RoboDK station: reto.rdk

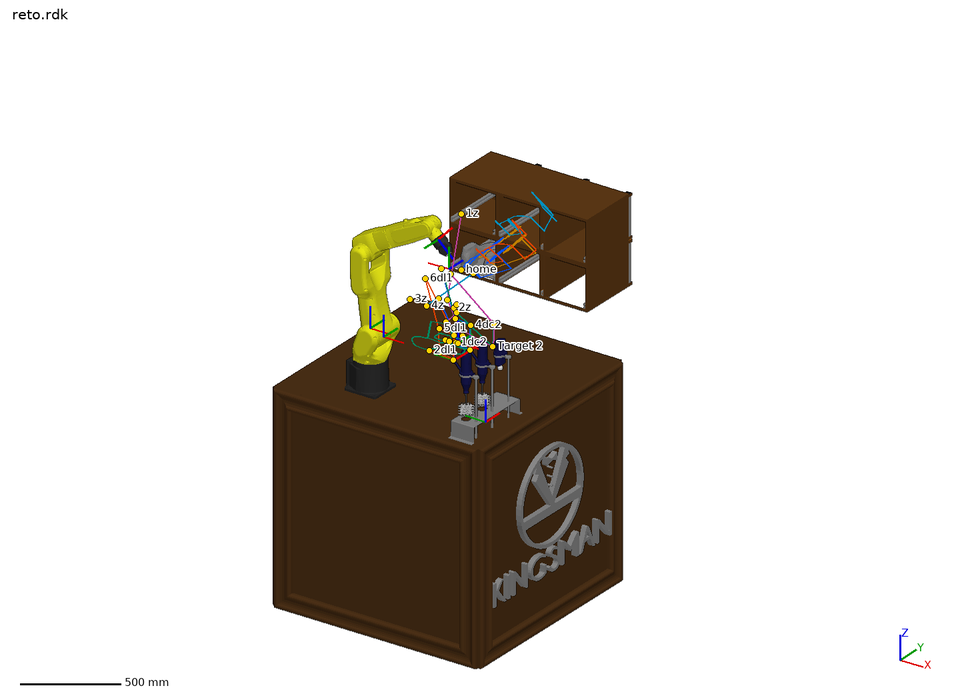
[picture v0: the station drawn from its stored meshes, robots at their saved joint values, targets as dots, program paths as lines]
Station reto (saved by RoboDK 5.5.4). Poses are relative to the parent item; angles as X-Y-Z fixed-axis rotations.
  - frame Fanuc LR Mate 200iD/7L Base at (0, 670, 330) mm
    - robot Fanuc LR Mate 200iD/7L: 6 axes, payload 7 kg, reach 911 mm, repeatability 0.03 mm, weight 27 kg
        modified DH rows (alpha deg, a mm, theta deg, d mm): 0, 0, 0, 330; -90, 50, -90, 0; 0, 440, 0, 0; -90, 35, 0, 420; 90, 0, 0, 0; -90, 0, 0, 80
        base shift (0, 0, -330) mm
        joint limits [-170, -70, -70, -190, -115, -360] to [170, 145, 215, 190, 115, 360]; home [0, 0, 0, 0, 0, 0]; saved at [0, -7.035, 27.253, 0, -70.54, 0]
      - frame RobotiQ 2F-140 Gripper (Mechanism) Base at (0, 0, 0) mm
        - robot RobotiQ 2F-140 Gripper (Mechanism) (model RobotiQ 2F140): 1 axes, payload 5 kg
            joint limits [0] to [140]; home [140]; saved at [30]
          - tool Tool 1, TCP at (0, 0, 190) mm
        - target open (joint target) at (0, 0, 190) mm; joints [30] of RobotiQ 2F-140 Gripper (Mechanism)
        - target close (joint target) at (-70.03, -6.66, -1.07) mm, rotated rx -1.32 ry 1.53 rz 3.85 deg; joints [10] of RobotiQ 2F-140 Gripper (Mechanism)
    - target home (Cartesian target) at (550, 0, 475) mm, rotated rx -180 ry -46.71 rz 0 deg; joints [0, 3.939, 7.691, 0, -50.978, 0] of Fanuc LR Mate 200iD/7L
  - frame rack at (-170, 1590, 240) mm, rotated rx 90 ry 0 rz 180 deg
    - object FullRack (1) at (-810, 360, -320) mm, size 835 x 510 x 385.3 mm, geometry from FullRack (1).STEP
    - target 1z (Cartesian target) at (-358.1, 564.97, -403.2) mm, rotated rx -26.57 ry -40.12 rz 107.86 deg; joints [70, -7.04, 27.25, 0, -70.54, 0] of Fanuc LR Mate 200iD/7L
    - target 2z (Cartesian target) at (-342.39, 58.73, -444.89) mm, rotated rx 2.43 ry -28.49 rz 101.39 deg; joints [48.708, 3.516, -60.085, -111.282, -47, 134.319] of Fanuc LR Mate 200iD/7L
    - target 3z (Cartesian target) at (-104.58, 56.68, -482.72) mm, rotated rx 2.43 ry -28.49 rz 101.39 deg; joints [97.474, -14.415, -55.536, -177.531, -28.246, 164.28] of Fanuc LR Mate 200iD/7L
    - target 4z (Cartesian target) at (-165.76, 16.78, -430.34) mm, rotated rx 2.43 ry -28.49 rz 101.39 deg; joints [82.687, 5.107, -71.647, -159.69, -45.234, 158.787] of Fanuc LR Mate 200iD/7L
    - target 5z (Cartesian target) at (-150, 20, 0) mm, rotated rx 2.43 ry -28.49 rz 101.39 deg; joints [88.603, 43.78, -43.517, 30.239, 18.18, -38.415] of Fanuc LR Mate 200iD/7L
    - target subida charola (Cartesian target) at (-343.88, 69.1, -423.53) mm, rotated rx 2.43 ry -28.49 rz 101.39 deg; joints [50.933, 3.87, -57.639, 68.607, 45.039, -48.263] of Fanuc LR Mate 200iD/7L
  - frame base herramental at (710, 650, 20) mm, rotated rx 0 ry 0 rz 90 deg
    - object Soporte de herramientas at (0, 0, 70) mm, rotated rx 90 ry 0 rz 180 deg, size 443.6 x 340 x 140 mm, geometry from Soporte de herramientas.STEP
  - frame dremel2 at (620, 650, 390) mm, rotated rx 0 ry 0 rz 90 deg
    - target 1dc2 (Cartesian target) at (0.49, 88.9, 17.55) mm, rotated rx -180 ry -61.75 rz -90 deg; joints [89.913, -3.297, -48.984, 180.078, 102.766, 0.058] of Fanuc LR Mate 200iD/7L
    - target 2dc2 (Cartesian target) at (0, 151.76, 13.3) mm, rotated rx -180 ry -61.75 rz -90 deg; joints [-4.961, -25.961, -32.248, 48.26, 5.86, -45.758] of Fanuc LR Mate 200iD/7L
    - target 3dc2 (Cartesian target) at (0, 4.92, 1.2) mm, rotated rx -180 ry -49.6 rz -90 deg; joints [-2.796, -1.172, -33.671, 162.466, 7.084, -160.778] of Fanuc LR Mate 200iD/7L
    - target 4dc2 (Cartesian target) at (0, 0.76, 138.38) mm, rotated rx -180 ry -49.6 rz -90 deg; joints [-2.768, -6.859, -13.429, 175.365, 27.075, -174.076] of Fanuc LR Mate 200iD/7L
    - target 5dc2 (Cartesian target) at (0, 92.68, 148.84) mm, rotated rx -180 ry -44.51 rz -90 deg; joints [-3.386, -17.516, -7.24, 176.175, 38.363, -174.583] of Fanuc LR Mate 200iD/7L
    - target 6dc2 (Cartesian target) at (477.83, 510, 116.81) mm, rotated rx -180 ry -49.6 rz 3.55 deg; joints [64.081, -25.306, -11.026, 143.659, 39.225, -130.203] of Fanuc LR Mate 200iD/7L
  - frame dremel1 at (620, 510.31, 389.97) mm, rotated rx 0 ry 0 rz 90 deg
    - target 1dl1 (Cartesian target) at (0.49, 88.9, 17.55) mm, rotated rx -180 ry -61.75 rz -90 deg; joints [-28.495, -9.165, -37.687, 76.78, 25.575, -60.993] of Fanuc LR Mate 200iD/7L
    - target 2dl1 (Cartesian target) at (0, 151.76, 13.3) mm, rotated rx -180 ry -61.75 rz -90 deg; joints [-34.725, -17.114, -36.143, 84.899, 30.251, -65.939] of Fanuc LR Mate 200iD/7L
    - target 3dl1 (Cartesian target) at (0, 4.92, 1.2) mm, rotated rx -180 ry -49.6 rz -90 deg; joints [-21.306, 2.651, -33.616, 117.955, 18.257, -105.014] of Fanuc LR Mate 200iD/7L
    - target 4dl1 (Cartesian target) at (0, 0.76, 138.38) mm, rotated rx -180 ry -48.03 rz -90 deg; joints [-20.886, -2.493, -13.042, 151.816, 34.141, -141.769] of Fanuc LR Mate 200iD/7L
    - target 5dl1 (Cartesian target) at (0, 92.68, 148.84) mm, rotated rx -180 ry -49.6 rz -90 deg; joints [-26.4, -14.504, -10.508, 146.56, 37.916, -134.648] of Fanuc LR Mate 200iD/7L
    - target 6dl1 (Cartesian target) at (477.83, 510, 116.81) mm, rotated rx -180 ry -55.33 rz 3.55 deg; joints [37.94, -45.517, -1.764, 129.234, 61.201, -109.727] of Fanuc LR Mate 200iD/7L
    - object cepillo1 at (0, -70, -50) mm, rotated rx 90 ry 0 rz 180 deg, size 80 x 351.1 x 124.1 mm, geometry from Dremel con brida.STEP
  - frame bote cera at (140, 586, 355) mm
    - target Target 1 (Cartesian target) at (316.19, 84, 136.54) mm, rotated rx -180 ry -46.71 rz 0 deg; joints [0, -28.492, -10.215, 0, -33.072, 0] of Fanuc LR Mate 200iD/7L
    - target Target 3 (Cartesian target) at (300.65, 202.07, 136.5) mm, rotated rx -180 ry -46.9 rz 15 deg; joints [15, -28.576, -10.266, 0, -32.834, 0] of Fanuc LR Mate 200iD/7L
    - target Target 2 (Cartesian target) at (513.63, 208.92, 6.17) mm, rotated rx -180 ry -50.56 rz 10.82 deg; joints [10.82, 7.34, -38.44, 0, -1, 0] of Fanuc LR Mate 200iD/7L
    - target Target 4 (Cartesian target) at (516.39, 216.06, 127.59) mm, rotated rx -179.95 ry -49.71 rz 10.96 deg; joints [11.533, 0.978, -20.278, 1.139, -20.021, -1.442] of Fanuc LR Mate 200iD/7L
    - target Target 5 (Cartesian target) at (-30, 622.41, 89.17) mm, rotated rx -179.99 ry -46.7 rz 79.99 deg; joints [77.59, -12.853, -22.678, -4.973, -20.717, 6.303] of Fanuc LR Mate 200iD/7L
  - program open (3 instructions, listed below)
  - program close (3 instructions, listed below)
  - program home (4 instructions, listed below)
  - object mesa at (-1220, 1130, 330) mm, size 1277.5 x 1274.9 x 1205 mm, geometry from mesa.STEP
  - frame zapato at (110, 1270, 40) mm
    - target Target 1 (Cartesian target) at (78.1, -83.2, 764.97) mm, rotated rx -180 ry -46.71 rz 70 deg; joints [70, -7.04, 27.25, 0, -70.54, 0] of Fanuc LR Mate 200iD/7L
    - target Target 2 (Cartesian target) at (48.8, -163.69, 316.74) mm, rotated rx 180 ry -45.09 rz 70 deg; joints [70, -19.91, -32.531, 0, -12.378, 0] of Fanuc LR Mate 200iD/7L
    - target Target 3 (Cartesian target) at (51.99, -36.78, 68.56) mm, rotated rx -154.66 ry -59.5 rz 70 deg; joints [58.654, 42.845, -90.321, 40.028, 62.94, -13.915] of Fanuc LR Mate 200iD/7L
    - target Target 4 (Cartesian target) at (0, 0, 0) mm, rotated rx -154.66 ry -59.5 rz 70 deg; joints [67.996, 54.587, -97.1, 29.193, 68.847, -10.257] of Fanuc LR Mate 200iD/7L
    - target Target 5 (Cartesian target) at (-12.96, -146.91, 298.71) mm, rotated rx -168.48 ry -59.46 rz 67.92 deg; joints [74.53, -18.6, -45.29, -158.86, -16.3, 156.27] of Fanuc LR Mate 200iD/7L
    - target Target 6 (Cartesian target) at (14.48, -93.65, 48.92) mm, rotated rx -154.66 ry -59.5 rz 70 deg; joints [59.102, 46.97, -102.654, -143.53, -72.674, 174.279] of Fanuc LR Mate 200iD/7L
  - program recoger cepillo cera (10 instructions, listed below)
  - program reset (1 instructions, listed below)
  - program recoger cepillo limpieza (10 instructions, listed below)
  - program recoger cera (9 instructions, listed below)
  - program pick charola (8 instructions, listed below)
  - program c1 recoger (7 instructions, listed below)
  - program c1 entregar (7 instructions, listed below)
  - program poscharolamesa (7 instructions, listed below)
  - program dejar cepillo limpieza (9 instructions, listed below)
  - program dejar cepillo cera (10 instructions, listed below)
  - program dejar  cera (9 instructions, listed below)
  - program rutinac1 (22 instructions, listed below)
  - machining project parribaizq: rotZ(0) | rotX(0)*rotY(0) | onStart | onPathStart | onApproach | onPoint | onRetract | onFinish | SetRPM(%1) | SetTool(%1) | Extruder(%1) | default | default | OutOnMov(%1) | OutOffMov(%1) | onPathFinish | M_RunCode(%1)
  - program platizq (163 instructions, listed below)
  - machining project plateralesizq: rotZ(0) | rotX(0)*rotY(0) | onStart | onPathStart | onApproach | onPoint | onRetract | onFinish | SetRPM(%1) | SetTool(%1) | Extruder(%1) | default | default | OutOnMov(%1) | OutOffMov(%1) | onPathFinish | M_RunCode(%1)
  - program parrizq (66 instructions, listed below)
  - machining project Path3 ajustes: rotZ(0) | rotX(0)*rotY(0) | onStart | onPathStart | onApproach | onPoint | onRetract | onFinish | SetRPM(%1) | SetTool(%1) | Extruder(%1) | default | default | OutOnMov(%1) | OutOffMov(%1) | onPathFinish | M_RunCode(%1)
  - program platder (154 instructions, listed below)
  - machining project Path4 ajustes: rotZ(0) | rotX(0)*rotY(0) | onStart | onPathStart | onApproach | onPoint | onRetract | onFinish | SetRPM(%1) | SetTool(%1) | Extruder(%1) | default | default | OutOnMov(%1) | OutOffMov(%1) | onPathFinish | M_RunCode(%1)
  - program parrder (59 instructions, listed below)
  - object zapatoconcharola at (-21.13, 1591.46, 262.04) mm, rotated rx 0 ry 0 rz -0.01 deg, size 250 x 350 x 100.5 mm, geometry from zapatoconcharola.STEP
    - object Ruta_IZQ at (-60, 470, 60) mm, rotated rx 0 ry 0 rz -90 deg, geometry from Curva importada
    - object R7 at (-105, 460, 60) mm, rotated rx 0 ry 0 rz -90 deg
  - object cepillo2 at (690, 650, 340) mm, rotated rx 90 ry 0 rz -90 deg, size 80 x 351.1 x 124.1 mm, geometry from Dremel con brida.STEP
  - machining project Path5 ajustes: rotZ(0) | rotX(0)*rotY(0) | onStart | onPathStart | onApproach | onPoint | onRetract | onFinish | SetRPM(%1) | SetTool(%1) | Extruder(%1) | default | default | OutOnMov(%1) | OutOffMov(%1) | onPathFinish | M_RunCode(%1)
  - program Path5 (163 instructions, listed below)
  - object Bote con brida at (698, 771, 410) mm, rotated rx 90 ry 0 rz -90 deg, size 75 x 160 x 85 mm, geometry from Bote con brida.STEP
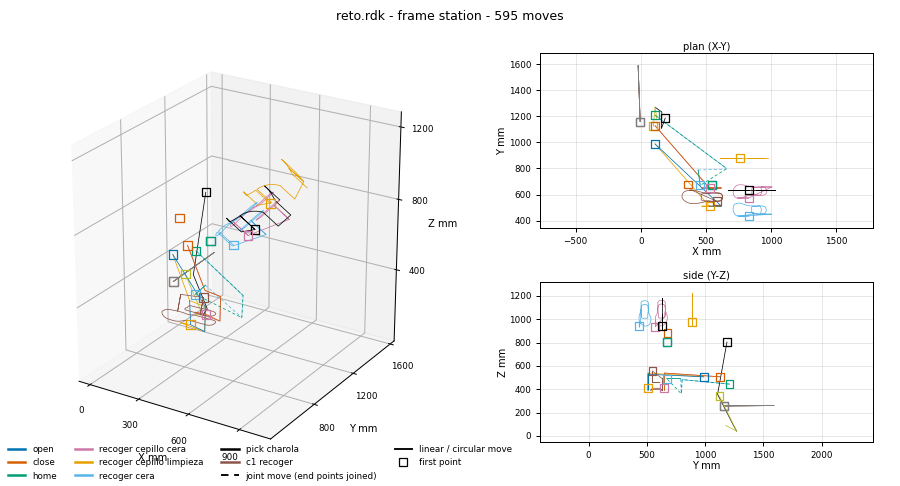
[picture p0: tool path of reto.rdk in frame station, 595 of 595 moves have a stored position in this frame; points joined in program order, loops and branches not executed]

--- program open (robot RobotiQ 2F-140 Gripper (Mechanism)) ---
  Est. Ref.: RobotiQ 2F-140 Gripper (Mechanism) Base
  Est. herr: Tool 1
  MoveJ (open)

--- program close (robot RobotiQ 2F-140 Gripper (Mechanism)) ---
  Est. Ref.: RobotiQ 2F-140 Gripper (Mechanism) Base
  Est. herr: Tool 1
  MoveJ (close)

--- program home (robot Fanuc LR Mate 200iD/7L) ---
  Est. Ref.: Fanuc LR Mate 200iD/7L Base
  MoveJ (home)
  Llamar open
  Separar de Tool 1

--- program recoger cepillo cera (robot Fanuc LR Mate 200iD/7L) ---
  Est. Ref.: dremel2
  Est. herr: Tool 1
  MoveL (1dc2)
  MoveL (Target 2) -> target 2dc2
  MoveL (Target 3) -> target 3dc2
  Llamar close
  Adjuntar a Tool 1
  MoveL (Target 4) -> target 4dc2
  MoveL (Target 5) -> target 5dc2
  MoveL (6dc2)

--- program reset (robot Fanuc LR Mate 200iD/7L) ---
  Reemplazar objetos

--- program recoger cepillo limpieza (robot Fanuc LR Mate 200iD/7L) ---
  Est. Ref.: dremel1
  Est. herr: Tool 1
  MoveL (1dl1)
  MoveL (2dl1)
  MoveL (3dl1)
  Adjuntar a Tool 1
  Llamar close
  MoveL (4dl1)
  MoveL (5dl1)
  MoveL (6dl1)

--- program recoger cera (robot Fanuc LR Mate 200iD/7L) ---
  Est. Ref.: bote cera
  Est. herr: Tool 1
  MoveJ (Target 1)
  MoveL (Target 3)
  MoveJ (Target 2)
  Llamar close
  Adjuntar a Tool 1
  MoveJ (Target 4)
  MoveL (Target 5)

--- program pick charola (robot Fanuc LR Mate 200iD/7L) ---
  Est. Ref.: zapato
  Est. herr: Tool 1
  MoveJ (Target 1)
  MoveL (Target 2)
  MoveL (Target 3)
  MoveL (Target 4)
  Llamar close
  Adjuntar a Tool 1

--- program c1 recoger (robot Fanuc LR Mate 200iD/7L) ---
  Est. Ref.: rack
  Est. herr: Tool 1
  MoveL (4z)
  MoveL (Target 4) -> target 5z
  Adjuntar a Tool 1
  Llamar close
  MoveL (4z)

--- program c1 entregar (robot Fanuc LR Mate 200iD/7L) ---
  Est. Ref.: rack
  Est. herr: Tool 1
  MoveL (4z)
  MoveL (Target 4) -> target 5z
  Separar de Tool 1
  Llamar open
  MoveL (4z)

--- program poscharolamesa (robot Fanuc LR Mate 200iD/7L) ---
  Est. Ref.: zapato
  Est. herr: Tool 1
  MoveJ (Target 5)
  MoveL (Target 4)
  Separar de Tool 1
  Llamar open
  MoveL (Target 6)

--- program dejar cepillo limpieza (robot Fanuc LR Mate 200iD/7L) ---
  Est. Ref.: dremel1
  Est. herr: Tool 1
  MoveL (6dl1)
  MoveL (4dl1)
  MoveL (3dl1)
  Separar de Tool 1
  Llamar open
  MoveL (1dl1)
  MoveL (5dl1)

--- program dejar cepillo cera (robot Fanuc LR Mate 200iD/7L) ---
  Est. Ref.: dremel2
  Est. herr: Tool 1
  MoveL (6dc2)
  MoveL (Target 5) -> target 5dc2
  MoveL (Target 4) -> target 4dc2
  MoveL (Target 3) -> target 3dc2
  Llamar open
  Separar de Tool 1
  MoveL (1dc2)
  MoveL (Target 2) -> target 2dc2

--- program dejar  cera (robot Fanuc LR Mate 200iD/7L) ---
  Est. Ref.: bote cera
  Est. herr: Tool 1
  MoveL (Target 5)
  MoveJ (Target 4)
  MoveJ (Target 2)
  Llamar open
  Separar de Tool 1
  MoveJ (Target 1)
  MoveL (Target 3)

--- program rutinac1 (robot Fanuc LR Mate 200iD/7L) ---
  Llamar home
  Llamar c1 recoger
  Llamar poscharolamesa
  Llamar home
  Llamar recoger cera
  Llamar recoger cepillo cera
  Llamar platizq
  Llamar parrizq
  Llamar platder
  Llamar parrder
  Llamar dejar cepillo cera
  Llamar recoger cepillo limpi...: recoger cepillo limpieza
  Llamar platizq
  Llamar parrizq
  Llamar platder
  Llamar parrder
  Llamar dejar cepillo limpieza
  Llamar Program1
  Llamar pick charola
  Llamar pos entrega
  Llamar c1 entregar
  Llamar home

--- program platizq (robot Fanuc LR Mate 200iD/7L) ---
  Suave(1)
  Establecer velocidad (1000.0 mm/s)
  Est. Ref.: RobotiQ 2F-140 Gripper (Mechanism) Base
  Est. herr: Tool 1
  Mostrar Tool 1
  MoveJ 1 to (286.31, 96.93, 301.9) mm, rotated rx 164.21 ry -43.9 rz -78.89 deg; joints [65.752, 52.412, -5.749, -44.813, -95.376, 119.1]
  MoveL 2 to (286.31, 96.93, 301.9) mm, rotated rx 164.21 ry -43.9 rz -78.89 deg; joints [65.752, 52.412, -5.749, -44.813, -95.376, 119.1]
  MoveL 3 to (266.7, 96.93, 203.84) mm, rotated rx 164.21 ry -43.9 rz -78.89 deg; joints [66.303, 57.855, -14.466, -44.7, -88.799, 124.852]
  MoveL 4 to (266.7, 96.93, 203.84) mm, rotated rx 164.21 ry -43.9 rz -78.89 deg; joints [66.303, 57.855, -14.466, -44.7, -88.799, 124.852]
  Establecer velocidad (50.0 mm/s)
  MoveL 5 to (278.42, 97.92, 203.84) mm, rotated rx 164.21 ry -43.9 rz -78.89 deg; joints [65.914, 55.94, -16.17, -44.64, -87.851, 126.317]
  MoveL 6 to (290.23, 97.9, 203.84) mm, rotated rx 164.21 ry -43.9 rz -78.89 deg; joints [65.577, 54.073, -17.804, -44.604, -86.914, 127.696]
  MoveL 7 to (301.99, 96.89, 203.84) mm, rotated rx 164.21 ry -43.9 rz -78.89 deg; joints [65.297, 52.255, -19.368, -44.595, -85.987, 128.985]
  MoveL 8 to (313.58, 94.89, 203.84) mm, rotated rx 164.21 ry -43.9 rz -78.89 deg; joints [65.079, 50.491, -20.859, -44.613, -85.069, 130.182]
  MoveL 9 to (324.92, 91.93, 204.39) mm, rotated rx 164.21 ry -43.9 rz -78.89 deg; joints [64.926, 48.755, -22.224, -44.657, -84.197, 131.247]
  MoveL 10 to (336.63, 87.99, 206.05) mm, rotated rx 164.21 ry -43.9 rz -78.89 deg; joints [64.822, 46.928, -23.474, -44.719, -83.376, 132.199]
  MoveL 11 to (348.23, 84.53, 208.85) mm, rotated rx 164.21 ry -43.9 rz -78.89 deg; joints [64.687, 45.145, -24.49, -44.762, -82.742, 133.009]
  MoveL 12 to (359.72, 81.7, 212.77) mm, rotated rx 164.21 ry -43.9 rz -78.89 deg; joints [64.506, 43.399, -25.277, -44.774, -82.298, 133.685]
  MoveL 13 to (371.38, 79.44, 216.26) mm, rotated rx 164.21 ry -43.9 rz -78.89 deg; joints [64.274, 41.719, -26.039, -44.769, -81.905, 134.376]
  MoveL 14 to (383.33, 77.72, 218.59) mm, rotated rx 164.21 ry -43.9 rz -78.89 deg; joints [63.986, 40.127, -26.87, -44.752, -81.496, 135.153]
  MoveL 15 to (395.57, 76.59, 219.75) mm, rotated rx 164.21 ry -43.9 rz -78.89 deg; joints [63.637, 38.623, -27.777, -44.724, -81.07, 136.022]
  MoveL 16 to (408.89, 76.07, 219.88) mm, rotated rx 164.21 ry -43.9 rz -78.89 deg; joints [63.191, 37.12, -28.809, -44.675, -80.612, 137.04]
  MoveL 17 to (422.22, 76.27, 219.88) mm, rotated rx 164.21 ry -43.9 rz -78.89 deg; joints [62.676, 35.694, -29.78, -44.591, -80.237, 138.056]
  MoveL 18 to (435.55, 76.27, 219.88) mm, rotated rx 164.21 ry -43.9 rz -78.89 deg; joints [62.158, 34.286, -30.714, -44.501, -79.885, 139.045]
  MoveL 19 to (448.88, 76.27, 219.88) mm, rotated rx 164.21 ry -43.9 rz -78.89 deg; joints [61.622, 32.904, -31.606, -44.396, -79.57, 140.012]
  MoveL 20 to (462.2, 76.27, 219.88) mm, rotated rx 164.21 ry -43.9 rz -78.89 deg; joints [61.067, 31.545, -32.457, -44.276, -79.291, 140.96]
  MoveL 21 to (470.53, 76.27, 219.88) mm, rotated rx 164.21 ry -43.9 rz -78.89 deg; joints [60.709, 30.706, -32.969, -44.192, -79.133, 141.543]
  MoveL 22 to (478.87, 76.27, 219.88) mm, rotated rx 164.21 ry -43.9 rz -78.89 deg; joints [60.344, 29.875, -33.467, -44.101, -78.989, 142.119]
  MoveL 23 to (487.2, 76.27, 219.88) mm, rotated rx 164.21 ry -43.9 rz -78.89 deg; joints [59.97, 29.052, -33.95, -44.003, -78.858, 142.689]
  MoveL 24 to (495.6, 76.03, 219.88) mm, rotated rx 164.21 ry -43.9 rz -78.89 deg; joints [59.603, 28.214, -34.431, -43.906, -78.722, 143.252]
  MoveL 25 to (501.43, 74.59, 219.88) mm, rotated rx 164.21 ry -43.9 rz -78.89 deg; joints [59.445, 27.564, -34.797, -43.886, -78.549, 143.607]
  MoveL 26 to (507.05, 71.76, 219.88) mm, rotated rx 164.21 ry -43.9 rz -78.89 deg; joints [59.406, 26.856, -35.188, -43.924, -78.289, 143.907]
  MoveL 27 to (511.98, 67.62, 219.88) mm, rotated rx 164.21 ry -43.9 rz -78.89 deg; joints [59.506, 26.142, -35.574, -44.026, -77.955, 144.121]
  MoveL 28 to (515.8, 62.47, 219.88) mm, rotated rx 164.21 ry -43.9 rz -78.89 deg; joints [59.745, 25.481, -35.925, -44.188, -77.568, 144.228]
  MoveL 29 to (518.26, 56.77, 219.88) mm, rotated rx 164.21 ry -43.9 rz -78.89 deg; joints [60.1, 24.923, -36.215, -44.397, -77.16, 144.226]
  MoveL 30 to (519.36, 50.99, 219.88) mm, rotated rx 164.21 ry -43.9 rz -78.89 deg; joints [60.532, 24.497, -36.433, -44.631, -76.76, 144.128]
  MoveL 31 to (519.45, 45.42, 219.88) mm, rotated rx 164.21 ry -43.9 rz -78.89 deg; joints [61, 24.185, -36.591, -44.872, -76.383, 143.967]
  MoveL 32 to (519.45, 39.87, 219.88) mm, rotated rx 164.21 ry -43.9 rz -78.89 deg; joints [61.476, 23.887, -36.74, -45.116, -76.008, 143.798]
  MoveL 33 to (518.9, 34.19, 219.88) mm, rotated rx 164.21 ry -43.9 rz -78.89 deg; joints [61.991, 23.64, -36.863, -45.373, -75.629, 143.588]
  MoveL 34 to (517.05, 28.4, 219.88) mm, rotated rx 164.21 ry -43.9 rz -78.89 deg; joints [62.579, 23.523, -36.921, -45.651, -75.253, 143.29]
  MoveL 35 to (513.81, 22.95, 219.88) mm, rotated rx 164.21 ry -43.9 rz -78.89 deg; joints [63.202, 23.567, -36.898, -45.928, -74.911, 142.915]
  MoveL 36 to (509.33, 18.32, 219.88) mm, rotated rx 164.21 ry -43.9 rz -78.89 deg; joints [63.805, 23.785, -36.791, -46.178, -74.638, 142.487]
  MoveL 37 to (503.95, 14.89, 219.88) mm, rotated rx 164.21 ry -43.9 rz -78.89 deg; joints [64.336, 24.157, -36.605, -46.377, -74.459, 142.042]
  MoveL 38 to (498.15, 12.84, 219.88) mm, rotated rx 164.21 ry -43.9 rz -78.89 deg; joints [64.757, 24.644, -36.358, -46.512, -74.384, 141.614]
  MoveL 39 to (490.56, 12.13, 219.88) mm, rotated rx 164.21 ry -43.9 rz -78.89 deg; joints [65.128, 25.38, -35.977, -46.596, -74.428, 141.114]
  MoveL 40 to (483.15, 12.13, 219.88) mm, rotated rx 164.21 ry -43.9 rz -78.89 deg; joints [65.422, 26.134, -35.578, -46.642, -74.529, 140.643]
  MoveL 41 to (475.75, 12.13, 219.88) mm, rotated rx 164.21 ry -43.9 rz -78.89 deg; joints [65.71, 26.891, -35.168, -46.682, -74.64, 140.166]
  MoveL 42 to (468.34, 12.13, 219.88) mm, rotated rx 164.21 ry -43.9 rz -78.89 deg; joints [65.992, 27.653, -34.747, -46.717, -74.761, 139.684]
  MoveL 43 to (460.94, 12.13, 219.88) mm, rotated rx 164.21 ry -43.9 rz -78.89 deg; joints [66.268, 28.419, -34.314, -46.745, -74.892, 139.196]
  MoveL 44 to (453.53, 12.13, 219.88) mm, rotated rx 164.21 ry -43.9 rz -78.89 deg; joints [66.537, 29.189, -33.869, -46.768, -75.034, 138.702]
  MoveL 45 to (438.87, 12.13, 219.88) mm, rotated rx 164.21 ry -43.9 rz -78.89 deg; joints [67.055, 30.73, -32.954, -46.798, -75.346, 137.706]
  MoveL 46 to (424.21, 12.13, 219.88) mm, rotated rx 164.21 ry -43.9 rz -78.89 deg; joints [67.551, 32.293, -31.991, -46.81, -75.7, 136.685]
  MoveL 47 to (409.55, 11.64, 219.88) mm, rotated rx 164.21 ry -43.9 rz -78.89 deg; joints [68.066, 33.859, -30.992, -46.82, -76.064, 135.624]
  MoveL 48 to (394.97, 10.16, 219.72) mm, rotated rx 164.21 ry -43.9 rz -78.89 deg; joints [68.635, 35.412, -29.992, -46.848, -76.39, 134.528]
  MoveL 49 to (382.83, 8.14, 218.52) mm, rotated rx 164.21 ry -43.9 rz -78.89 deg; joints [69.153, 36.756, -29.261, -46.901, -76.56, 133.663]
  MoveL 50 to (370.99, 5.48, 216.16) mm, rotated rx 164.21 ry -43.9 rz -78.89 deg; joints [69.696, 38.124, -28.661, -46.982, -76.623, 132.878]
  MoveL 51 to (359.45, 2.34, 212.67) mm, rotated rx 164.21 ry -43.9 rz -78.89 deg; joints [70.252, 39.521, -28.181, -47.084, -76.593, 132.175]
  MoveL 52 to (347.95, -0.34, 208.77) mm, rotated rx 164.21 ry -43.9 rz -78.89 deg; joints [70.757, 40.975, -27.691, -47.163, -76.599, 131.494]
  MoveL 53 to (336.16, -2.45, 205.96) mm, rotated rx 164.21 ry -43.9 rz -78.89 deg; joints [71.214, 42.455, -26.991, -47.186, -76.778, 130.683]
  MoveL 54 to (324.08, -3.96, 204.31) mm, rotated rx 164.21 ry -43.9 rz -78.89 deg; joints [71.621, 43.967, -26.069, -47.154, -77.137, 129.734]
  MoveL 55 to (313.03, -4.77, 203.84) mm, rotated rx 164.21 ry -43.9 rz -78.89 deg; joints [71.942, 45.354, -25.048, -47.081, -77.619, 128.766]
  MoveL 56 to (301.89, -5.05, 203.84) mm, rotated rx 164.21 ry -43.9 rz -78.89 deg; joints [72.219, 46.792, -23.9, -46.979, -78.218, 127.731]
  MoveL 57 to (290.76, -5.05, 203.84) mm, rotated rx 164.21 ry -43.9 rz -78.89 deg; joints [72.468, 48.29, -22.683, -46.865, -78.882, 126.664]
  MoveL 58 to (279.63, -4.45, 203.84) mm, rotated rx 164.21 ry -43.9 rz -78.89 deg; joints [72.67, 49.87, -21.378, -46.736, -79.639, 125.566]
  MoveL 59 to (268.65, -2.57, 203.84) mm, rotated rx 164.21 ry -43.9 rz -78.89 deg; joints [72.775, 51.554, -19.963, -46.582, -80.538, 124.452]
  MoveL 60 to (257.97, 0.55, 204.05) mm, rotated rx 164.21 ry -43.9 rz -78.89 deg; joints [72.788, 53.327, -18.42, -46.409, -81.592, 123.311]
  MoveL 61 to (247.78, 4.86, 204.72) mm, rotated rx 164.21 ry -43.9 rz -78.89 deg; joints [72.712, 55.166, -16.728, -46.225, -82.813, 122.127]
  MoveL 62 to (238.11, 10.33, 205.8) mm, rotated rx 164.21 ry -43.9 rz -78.89 deg; joints [72.55, 57.095, -14.875, -46.041, -84.209, 120.891]
  MoveL 63 to (229.2, 16.81, 207.18) mm, rotated rx 164.21 ry -43.9 rz -78.89 deg; joints [72.312, 59.098, -12.887, -45.873, -85.758, 119.618]
  MoveL 64 to (224.26, 21.15, 208.1) mm, rotated rx 164.21 ry -43.9 rz -78.89 deg; joints [72.135, 60.344, -11.627, -45.784, -86.76, 118.833]
  MoveL 65 to (219.61, 25.82, 209.08) mm, rotated rx 164.21 ry -43.9 rz -78.89 deg; joints [71.932, 61.636, -10.307, -45.707, -87.823, 118.025]
  MoveL 66 to (215.3, 30.86, 210.08) mm, rotated rx 164.21 ry -43.9 rz -78.89 deg; joints [71.703, 62.982, -8.922, -45.646, -88.953, 117.192]
  MoveL 67 to (212.09, 36.67, 210.88) mm, rotated rx 164.21 ry -43.9 rz -78.89 deg; joints [71.405, 64.241, -7.632, -45.597, -90.066, 116.477]
  MoveL 68 to (210.42, 43.11, 211.32) mm, rotated rx 164.21 ry -43.9 rz -78.89 deg; joints [71.038, 65.263, -6.607, -45.556, -91.043, 115.999]
  MoveL 69 to (210.2, 50.56, 211.38) mm, rotated rx 164.21 ry -43.9 rz -78.89 deg; joints [70.581, 66.055, -5.845, -45.512, -91.901, 115.774]
  MoveL 70 to (210.79, 57.98, 211.23) mm, rotated rx 164.21 ry -43.9 rz -78.89 deg; joints [70.11, 66.669, -5.279, -45.469, -92.632, 115.699]
  MoveL 71 to (212.67, 65.14, 210.74) mm, rotated rx 164.21 ry -43.9 rz -78.89 deg; joints [69.628, 66.895, -5.129, -45.414, -93.08, 115.929]
  MoveL 72 to (215.78, 71.8, 209.97) mm, rotated rx 164.21 ry -43.9 rz -78.89 deg; joints [69.148, 66.715, -5.407, -45.341, -93.224, 116.463]
  MoveL 73 to (220.02, 77.81, 208.99) mm, rotated rx 164.21 ry -43.9 rz -78.89 deg; joints [68.681, 66.157, -6.073, -45.25, -93.086, 117.265]
  MoveL 74 to (225.23, 82.95, 207.91) mm, rotated rx 164.21 ry -43.9 rz -78.89 deg; joints [68.241, 65.29, -7.046, -45.149, -92.711, 118.264]
  MoveL 75 to (231.27, 87.1, 206.82) mm, rotated rx 164.21 ry -43.9 rz -78.89 deg; joints [67.839, 64.187, -8.237, -45.048, -92.152, 119.39]
  MoveL 76 to (237.96, 90.11, 205.82) mm, rotated rx 164.21 ry -43.9 rz -78.89 deg; joints [67.486, 62.919, -9.563, -44.956, -91.462, 120.575]
  MoveL 77 to (244.99, 92.39, 204.99) mm, rotated rx 164.21 ry -43.9 rz -78.89 deg; joints [67.165, 61.61, -10.891, -44.876, -90.744, 121.737]
  MoveL 78 to (252.12, 94.28, 204.38) mm, rotated rx 164.21 ry -43.9 rz -78.89 deg; joints [66.861, 60.337, -12.145, -44.808, -90.065, 122.832]
  MoveL 79 to (259.35, 95.8, 203.99) mm, rotated rx 164.21 ry -43.9 rz -78.89 deg; joints [66.574, 59.089, -13.334, -44.749, -89.419, 123.869]
  MoveL 80 to (266.7, 96.93, 203.84) mm, rotated rx 164.21 ry -43.9 rz -78.89 deg; joints [66.303, 57.855, -14.466, -44.7, -88.799, 124.852]
  Establecer velocidad (1000.0 mm/s)
  MoveL 81 to (266.7, 96.93, 203.84) mm, rotated rx 164.21 ry -43.9 rz -78.89 deg; joints [66.303, 57.855, -14.466, -44.7, -88.799, 124.852]
  MoveL 82 to (286.31, 96.93, 301.9) mm, rotated rx 164.21 ry -43.9 rz -78.89 deg; joints [65.752, 52.412, -5.749, -44.813, -95.376, 119.1]
  Establecer velocidad (1000.0 mm/s)
  MoveL 83 to (477.63, 11.95, 367.18) mm, rotated rx 164.21 ry -43.9 rz -78.89 deg; joints [65.653, 19.725, -16.781, -44.59, -87.591, 126.925]
  MoveL 84 to (458.02, 11.95, 269.13) mm, rotated rx 164.21 ry -43.9 rz -78.89 deg; joints [66.39, 25.861, -28.191, -45.767, -79.052, 134.582]
  MoveL 85 to (458.02, 11.95, 269.13) mm, rotated rx 164.21 ry -43.9 rz -78.89 deg; joints [66.39, 25.861, -28.191, -45.767, -79.052, 134.582]
  Establecer velocidad (50.0 mm/s)
  MoveL 86 to (478.18, 12.91, 269.13) mm, rotated rx 164.21 ry -43.9 rz -78.89 deg; joints [65.55, 23.716, -29.218, -45.608, -78.862, 135.856]
  MoveL 87 to (498.18, 15.71, 269.13) mm, rotated rx 164.21 ry -43.9 rz -78.89 deg; joints [64.505, 21.712, -30.109, -45.341, -78.885, 137.152]
  MoveL 88 to (504.68, 17.51, 269.13) mm, rotated rx 164.21 ry -43.9 rz -78.89 deg; joints [64.075, 21.114, -30.361, -45.21, -78.971, 137.601]
  MoveL 89 to (510.58, 20.71, 269.13) mm, rotated rx 164.21 ry -43.9 rz -78.89 deg; joints [63.541, 20.656, -30.55, -45.028, -79.164, 138.069]
  MoveL 90 to (515.69, 25.1, 269.13) mm, rotated rx 164.21 ry -43.9 rz -78.89 deg; joints [62.929, 20.352, -30.674, -44.804, -79.448, 138.537]
  MoveL 91 to (519.69, 30.53, 269.13) mm, rotated rx 164.21 ry -43.9 rz -78.89 deg; joints [62.273, 20.228, -30.724, -44.549, -79.809, 138.98]
  MoveL 92 to (522.14, 36.78, 269.13) mm, rotated rx 164.21 ry -43.9 rz -78.89 deg; joints [61.616, 20.319, -30.688, -44.279, -80.231, 139.364]
  MoveL 93 to (522.78, 43.44, 269.13) mm, rotated rx 164.21 ry -43.9 rz -78.89 deg; joints [61.012, 20.629, -30.562, -44.02, -80.683, 139.653]
  MoveL 94 to (522.59, 48.79, 269.13) mm, rotated rx 164.21 ry -43.9 rz -78.89 deg; joints [60.564, 20.956, -30.427, -43.822, -81.047, 139.84]
  MoveL 95 to (521.37, 53.92, 269.13) mm, rotated rx 164.21 ry -43.9 rz -78.89 deg; joints [60.188, 21.38, -30.25, -43.65, -81.4, 139.954]
  MoveL 96 to (519.11, 58.74, 269.13) mm, rotated rx 164.21 ry -43.9 rz -78.89 deg; joints [59.894, 21.894, -30.031, -43.507, -81.734, 139.987]
  MoveL 97 to (515.98, 62.98, 269.13) mm, rotated rx 164.21 ry -43.9 rz -78.89 deg; joints [59.694, 22.466, -29.782, -43.401, -82.034, 139.942]
  MoveL 98 to (512.14, 66.64, 269.13) mm, rotated rx 164.21 ry -43.9 rz -78.89 deg; joints [59.578, 23.076, -29.51, -43.328, -82.3, 139.827]
  MoveL 99 to (506.24, 70.37, 269.13) mm, rotated rx 164.21 ry -43.9 rz -78.89 deg; joints [59.557, 23.902, -29.133, -43.285, -82.588, 139.579]
  MoveL 100 to (499.6, 72.56, 269.13) mm, rotated rx 164.21 ry -43.9 rz -78.89 deg; joints [59.693, 24.715, -28.75, -43.306, -82.785, 139.227]
  MoveL 101 to (492.7, 73.71, 269.13) mm, rotated rx 164.21 ry -43.9 rz -78.89 deg; joints [59.921, 25.494, -28.372, -43.364, -82.922, 138.819]
  MoveL 102 to (485.76, 74.65, 269.13) mm, rotated rx 164.21 ry -43.9 rz -78.89 deg; joints [60.163, 26.269, -27.988, -43.427, -83.055, 138.397]
  MoveL 103 to (478.81, 75.37, 269.13) mm, rotated rx 164.21 ry -43.9 rz -78.89 deg; joints [60.417, 27.038, -27.597, -43.493, -83.184, 137.962]
  MoveL 104 to (471.83, 75.89, 269.13) mm, rotated rx 164.21 ry -43.9 rz -78.89 deg; joints [60.683, 27.801, -27.199, -43.563, -83.31, 137.513]
  MoveL 105 to (455.34, 76.31, 269.13) mm, rotated rx 164.21 ry -43.9 rz -78.89 deg; joints [61.352, 29.581, -26.237, -43.738, -83.593, 136.41]
  MoveL 106 to (438.86, 75.72, 269.13) mm, rotated rx 164.21 ry -43.9 rz -78.89 deg; joints [62.068, 31.335, -25.243, -43.922, -83.864, 135.25]
  MoveL 107 to (429.14, 74.68, 269.13) mm, rotated rx 164.21 ry -43.9 rz -78.89 deg; joints [62.528, 32.349, -24.648, -44.04, -84.002, 134.532]
  MoveL 108 to (419.56, 73.03, 269.13) mm, rotated rx 164.21 ry -43.9 rz -78.89 deg; joints [63.016, 33.327, -24.06, -44.166, -84.115, 133.8]
  MoveL 109 to (410.02, 71.52, 269.13) mm, rotated rx 164.21 ry -43.9 rz -78.89 deg; joints [63.482, 34.326, -23.446, -44.279, -84.258, 133.062]
  MoveL 110 to (400.32, 71.63, 269.13) mm, rotated rx 164.21 ry -43.9 rz -78.89 deg; joints [63.826, 35.453, -22.737, -44.343, -84.544, 132.337]
  MoveL 111 to (390.63, 71.78, 269.13) mm, rotated rx 164.21 ry -43.9 rz -78.89 deg; joints [64.158, 36.602, -21.997, -44.401, -84.858, 131.597]
  MoveL 112 to (380.93, 71.76, 269.13) mm, rotated rx 164.21 ry -43.9 rz -78.89 deg; joints [64.494, 37.763, -21.232, -44.458, -85.186, 130.835]
  MoveL 113 to (376.53, 71.63, 269.13) mm, rotated rx 164.21 ry -43.9 rz -78.89 deg; joints [64.653, 38.29, -20.879, -44.486, -85.335, 130.481]
  MoveL 114 to (372.12, 71.37, 269.13) mm, rotated rx 164.21 ry -43.9 rz -78.89 deg; joints [64.818, 38.815, -20.524, -44.516, -85.479, 130.12]
  MoveL 115 to (367.74, 70.93, 269.13) mm, rotated rx 164.21 ry -43.9 rz -78.89 deg; joints [64.995, 39.333, -20.17, -44.549, -85.616, 129.753]
  MoveL 116 to (363.46, 69.88, 269.13) mm, rotated rx 164.21 ry -43.9 rz -78.89 deg; joints [65.209, 39.807, -19.843, -44.594, -85.707, 129.379]
  MoveL 117 to (359.87, 67.33, 269.13) mm, rotated rx 164.21 ry -43.9 rz -78.89 deg; joints [65.504, 40.113, -19.631, -44.667, -85.663, 129.031]
  MoveL 118 to (357.66, 64.38, 269.13) mm, rotated rx 164.21 ry -43.9 rz -78.89 deg; joints [65.782, 40.224, -19.553, -44.742, -85.533, 128.79]
  MoveL 119 to (356.45, 60.9, 269.13) mm, rotated rx 164.21 ry -43.9 rz -78.89 deg; joints [66.066, 40.18, -19.584, -44.824, -85.323, 128.622]
  MoveL 120 to (356.53, 57.23, 269.13) mm, rotated rx 164.21 ry -43.9 rz -78.89 deg; joints [66.323, 39.963, -19.735, -44.905, -85.046, 128.555]
  MoveL 121 to (358.19, 51.95, 269.13) mm, rotated rx 164.21 ry -43.9 rz -78.89 deg; joints [66.647, 39.463, -20.08, -45.018, -84.586, 128.584]
  MoveL 122 to (359.99, 46.73, 269.13) mm, rotated rx 164.21 ry -43.9 rz -78.89 deg; joints [66.967, 38.954, -20.429, -45.132, -84.127, 128.62]
  MoveL 123 to (359.44, 44.38, 269.13) mm, rotated rx 164.21 ry -43.9 rz -78.89 deg; joints [67.153, 38.898, -20.467, -45.187, -83.977, 128.523]
  MoveL 124 to (358.75, 42.02, 269.13) mm, rotated rx 164.21 ry -43.9 rz -78.89 deg; joints [67.344, 38.861, -20.492, -45.242, -83.832, 128.414]
  MoveL 125 to (358.07, 39.66, 269.13) mm, rotated rx 164.21 ry -43.9 rz -78.89 deg; joints [67.535, 38.823, -20.518, -45.297, -83.687, 128.306]
  MoveL 126 to (357.4, 37.29, 269.13) mm, rotated rx 164.21 ry -43.9 rz -78.89 deg; joints [67.727, 38.785, -20.544, -45.352, -83.541, 128.198]
  MoveL 127 to (356.75, 34.93, 269.13) mm, rotated rx 164.21 ry -43.9 rz -78.89 deg; joints [67.918, 38.745, -20.571, -45.407, -83.395, 128.09]
  MoveL 128 to (356.37, 32.52, 269.13) mm, rotated rx 164.21 ry -43.9 rz -78.89 deg; joints [68.104, 38.67, -20.622, -45.463, -83.235, 128.004]
  MoveL 129 to (356.94, 27.7, 269.13) mm, rotated rx 164.21 ry -43.9 rz -78.89 deg; joints [68.439, 38.357, -20.834, -45.573, -82.863, 127.935]
  MoveL 130 to (359.06, 23.33, 269.13) mm, rotated rx 164.21 ry -43.9 rz -78.89 deg; joints [68.699, 37.876, -21.156, -45.674, -82.464, 127.996]
  MoveL 131 to (362.26, 19.68, 269.13) mm, rotated rx 164.21 ry -43.9 rz -78.89 deg; joints [68.877, 37.301, -21.538, -45.76, -82.078, 128.156]
  MoveL 132 to (366.48, 17.3, 269.13) mm, rotated rx 164.21 ry -43.9 rz -78.89 deg; joints [68.933, 36.666, -21.955, -45.818, -81.75, 128.421]
  MoveL 133 to (371.27, 16.51, 269.13) mm, rotated rx 164.21 ry -43.9 rz -78.89 deg; joints [68.854, 36.04, -22.361, -45.839, -81.52, 128.766]
  MoveL 134 to (376.12, 16.06, 269.13) mm, rotated rx 164.21 ry -43.9 rz -78.89 deg; joints [68.746, 35.43, -22.752, -45.85, -81.319, 129.12]
  MoveL 135 to (380.98, 15.85, 269.13) mm, rotated rx 164.21 ry -43.9 rz -78.89 deg; joints [68.618, 34.834, -23.128, -45.854, -81.141, 129.477]
  MoveL 136 to (385.85, 15.8, 269.13) mm, rotated rx 164.21 ry -43.9 rz -78.89 deg; joints [68.476, 34.25, -23.493, -45.854, -80.981, 129.833]
  MoveL 137 to (390.72, 15.85, 269.13) mm, rotated rx 164.21 ry -43.9 rz -78.89 deg; joints [68.324, 33.675, -23.848, -45.849, -80.834, 130.189]
  MoveL 138 to (396.17, 15.99, 269.13) mm, rotated rx 164.21 ry -43.9 rz -78.89 deg; joints [68.146, 33.04, -24.234, -45.84, -80.682, 130.585]
  MoveL 139 to (401.62, 16.18, 269.13) mm, rotated rx 164.21 ry -43.9 rz -78.89 deg; joints [67.961, 32.412, -24.61, -45.827, -80.54, 130.977]
  MoveL 140 to (407.07, 16.35, 269.13) mm, rotated rx 164.21 ry -43.9 rz -78.89 deg; joints [67.774, 31.789, -24.978, -45.813, -80.405, 131.365]
  MoveL 141 to (412.52, 16.47, 269.13) mm, rotated rx 164.21 ry -43.9 rz -78.89 deg; joints [67.589, 31.167, -25.34, -45.799, -80.273, 131.746]
  MoveL 142 to (417.87, 15.44, 269.13) mm, rotated rx 164.21 ry -43.9 rz -78.89 deg; joints [67.496, 30.507, -25.718, -45.815, -80.07, 132.081]
  MoveL 143 to (423.28, 14.13, 269.13) mm, rotated rx 164.21 ry -43.9 rz -78.89 deg; joints [67.421, 29.831, -26.097, -45.839, -79.854, 132.405]
  MoveL 144 to (429.21, 12.8, 269.13) mm, rotated rx 164.21 ry -43.9 rz -78.89 deg; joints [67.33, 29.099, -26.502, -45.862, -79.63, 132.758]
  MoveL 145 to (433.93, 12.19, 269.13) mm, rotated rx 164.21 ry -43.9 rz -78.89 deg; joints [67.22, 28.54, -26.805, -45.865, -79.491, 133.049]
  MoveL 146 to (437.62, 11.98, 269.13) mm, rotated rx 164.21 ry -43.9 rz -78.89 deg; joints [67.111, 28.118, -27.031, -45.858, -79.403, 133.283]
  MoveL 147 to (441.07, 11.95, 269.13) mm, rotated rx 164.21 ry -43.9 rz -78.89 deg; joints [66.994, 27.732, -27.235, -45.846, -79.336, 133.505]
  MoveL 148 to (444.06, 11.95, 269.13) mm, rotated rx 164.21 ry -43.9 rz -78.89 deg; joints [66.889, 27.399, -27.409, -45.834, -79.281, 133.698]
  MoveL 149 to (447.91, 11.95, 269.13) mm, rotated rx 164.21 ry -43.9 rz -78.89 deg; joints [66.754, 26.974, -27.629, -45.817, -79.214, 133.944]
  MoveL 150 to (452.73, 11.95, 269.13) mm, rotated rx 164.21 ry -43.9 rz -78.89 deg; joints [66.581, 26.442, -27.9, -45.795, -79.134, 134.25]
  MoveL 151 to (458.02, 11.95, 269.13) mm, rotated rx 164.21 ry -43.9 rz -78.89 deg; joints [66.39, 25.861, -28.191, -45.767, -79.052, 134.582]
  Establecer velocidad (1000.0 mm/s)
  MoveL 152 to (458.02, 11.95, 269.13) mm, rotated rx 164.21 ry -43.9 rz -78.89 deg; joints [66.39, 25.861, -28.191, -45.767, -79.052, 134.582]
  MoveL 153 to (477.63, 11.95, 367.18) mm, rotated rx 164.21 ry -43.9 rz -78.89 deg; joints [65.653, 19.725, -16.781, -44.59, -87.591, 126.925]

--- program parrizq (robot Fanuc LR Mate 200iD/7L) ---
  Suave(1)
  Establecer velocidad (1000.0 mm/s)
  Est. Ref.: RobotiQ 2F-140 Gripper (Mechanism) Base
  Est. herr: Tool 1
  Mostrar Tool 1
  MoveJ 1 to (272.96, -213.5, 226.79) mm, rotated rx 167.56 ry 24.48 rz -95.21 deg; joints [110.369, 49.011, -11.55, 27.852, -78.634, 61.476]
  MoveL 2 to (272.96, -213.5, 226.79) mm, rotated rx 167.56 ry 24.48 rz -95.21 deg; joints [110.369, 49.011, -11.55, 27.852, -78.634, 61.476]
  MoveL 3 to (253.35, -213.5, 128.73) mm, rotated rx 167.56 ry 24.48 rz -95.21 deg; joints [109.892, 55.363, -19.801, 28.933, -71.154, 57.834]
  MoveL 4 to (253.35, -213.5, 128.73) mm, rotated rx 167.56 ry 24.48 rz -95.21 deg; joints [109.892, 55.363, -19.801, 28.933, -71.154, 57.834]
  Establecer velocidad (50.0 mm/s)
  MoveL 5 to (243.62, -213.5, 127.58) mm, rotated rx 167.56 ry 24.48 rz -95.21 deg; joints [109.663, 56.96, -18.533, 28.742, -72.161, 58.678]
  MoveL 6 to (233.9, -213.5, 126.22) mm, rotated rx 167.56 ry 24.48 rz -95.21 deg; joints [109.439, 58.652, -17.188, 28.552, -73.239, 59.549]
  MoveL 7 to (223.13, -213.5, 124.47) mm, rotated rx 167.56 ry 24.48 rz -95.21 deg; joints [109.197, 60.658, -15.585, 28.341, -74.537, 60.557]
  MoveL 8 to (210.98, -213.5, 122.18) mm, rotated rx 167.56 ry 24.48 rz -95.21 deg; joints [108.93, 63.14, -13.582, 28.101, -76.181, 61.771]
  MoveL 9 to (200.56, -213.5, 119.96) mm, rotated rx 167.56 ry 24.48 rz -95.21 deg; joints [108.707, 65.515, -11.632, 27.894, -77.8, 62.908]
  MoveL 10 to (195.63, -213.5, 118.82) mm, rotated rx 167.56 ry 24.48 rz -95.21 deg; joints [108.603, 66.748, -10.603, 27.795, -78.663, 63.49]
  MoveL 11 to (191.25, -213.5, 117.76) mm, rotated rx 167.56 ry 24.48 rz -95.21 deg; joints [108.512, 67.922, -9.612, 27.706, -79.497, 64.041]
  MoveL 12 to (189.42, -213.5, 117.22) mm, rotated rx 167.56 ry 24.48 rz -95.21 deg; joints [108.474, 68.442, -9.179, 27.67, -79.864, 64.28]
  MoveL 13 to (188.23, -213.5, 116.45) mm, rotated rx 167.56 ry 24.48 rz -95.21 deg; joints [108.449, 68.797, -8.939, 27.65, -80.065, 64.414]
  MoveL 14 to (187.22, -213.5, 115.14) mm, rotated rx 167.56 ry 24.48 rz -95.21 deg; joints [108.429, 69.117, -8.805, 27.639, -80.175, 64.496]
  MoveL 15 to (186.8, -213.5, 113.88) mm, rotated rx 167.56 ry 24.48 rz -95.21 deg; joints [108.42, 69.27, -8.826, 27.641, -80.152, 64.494]
  MoveL 16 to (186.72, -213.5, 112.35) mm, rotated rx 167.56 ry 24.48 rz -95.21 deg; joints [108.418, 69.327, -8.979, 27.654, -80.016, 64.423]
  MoveL 17 to (186.72, -213.5, 110.28) mm, rotated rx 167.56 ry 24.48 rz -95.21 deg; joints [108.418, 69.375, -9.214, 27.673, -79.807, 64.312]
  MoveL 18 to (186.72, -213.5, 106.61) mm, rotated rx 167.56 ry 24.48 rz -95.21 deg; joints [108.418, 69.466, -9.625, 27.708, -79.443, 64.118]
  MoveL 19 to (186.72, -213.5, 102.35) mm, rotated rx 167.56 ry 24.48 rz -95.21 deg; joints [108.418, 69.58, -10.095, 27.75, -79.027, 63.896]
  MoveL 20 to (186.72, -213.5, 98.08) mm, rotated rx 167.56 ry 24.48 rz -95.21 deg; joints [108.419, 69.703, -10.557, 27.792, -78.619, 63.676]
  MoveL 21 to (186.72, -213.5, 93.7) mm, rotated rx 167.56 ry 24.48 rz -95.21 deg; joints [108.419, 69.839, -11.022, 27.837, -78.207, 63.455]
  Establecer velocidad (1000.0 mm/s)
  MoveL 22 to (186.72, -213.5, 93.7) mm, rotated rx 167.56 ry 24.48 rz -95.21 deg; joints [108.419, 69.839, -11.022, 27.837, -78.207, 63.455]
  MoveL 23 to (206.33, -213.5, 191.76) mm, rotated rx 167.56 ry 24.48 rz -95.21 deg; joints [108.829, 62.976, -4.24, 27.356, -84.408, 66.266]
  Establecer velocidad (1000.0 mm/s)
  MoveL 24 to (282.76, -213.5, 227.74) mm, rotated rx 167.56 ry 24.48 rz -95.21 deg; joints [110.616, 47.422, -12.667, 27.954, -77.76, 60.724]
  MoveL 25 to (263.15, -213.5, 129.69) mm, rotated rx 167.56 ry 24.48 rz -95.21 deg; joints [110.128, 53.835, -21.017, 29.125, -70.199, 57.004]
  MoveL 26 to (263.15, -213.5, 129.69) mm, rotated rx 167.56 ry 24.48 rz -95.21 deg; joints [110.128, 53.835, -21.017, 29.125, -70.199, 57.004]
  Establecer velocidad (50.0 mm/s)
  MoveL 27 to (281.65, -213.5, 132.2) mm, rotated rx 167.56 ry 24.48 rz -95.21 deg; joints [110.589, 51.077, -23.049, 29.466, -68.635, 55.544]
  MoveL 28 to (301.97, -213.5, 137.15) mm, rotated rx 167.56 ry 24.48 rz -95.21 deg; joints [111.118, 48.122, -24.824, 29.776, -67.331, 54.144]
  MoveL 29 to (321.64, -213.5, 144.29) mm, rotated rx 167.56 ry 24.48 rz -95.21 deg; joints [111.656, 45.275, -26.098, 29.995, -66.468, 52.996]
  MoveL 30 to (340.4, -213.5, 153.54) mm, rotated rx 167.56 ry 24.48 rz -95.21 deg; joints [112.194, 42.519, -26.892, 30.113, -66.022, 52.106]
  MoveL 31 to (358.05, -213.5, 164.78) mm, rotated rx 167.56 ry 24.48 rz -95.21 deg; joints [112.723, 39.856, -27.22, 30.127, -65.976, 51.48]
  MoveL 32 to (374.35, -213.5, 177.88) mm, rotated rx 167.56 ry 24.48 rz -95.21 deg; joints [113.234, 37.297, -27.095, 30.04, -66.311, 51.118]
  MoveL 33 to (389.14, -213.5, 192.68) mm, rotated rx 167.56 ry 24.48 rz -95.21 deg; joints [113.717, 34.864, -26.537, 29.863, -67.01, 51.015]
  Establecer velocidad (1000.0 mm/s)
  MoveL 34 to (389.14, -213.5, 192.68) mm, rotated rx 167.56 ry 24.48 rz -95.21 deg; joints [113.717, 34.864, -26.537, 29.863, -67.01, 51.015]
  MoveL 35 to (408.75, -213.5, 290.74) mm, rotated rx 167.56 ry 24.48 rz -95.21 deg; joints [114.386, 28.772, -16.112, 28.126, -76.436, 55.757]
  Establecer velocidad (1000.0 mm/s)
  MoveL 36 to (517.53, -213.5, 256.38) mm, rotated rx 167.56 ry 24.48 rz -95.21 deg; joints [118.847, 17.742, -25.712, 29.024, -69.993, 47.14]
  MoveL 37 to (497.92, -213.5, 158.32) mm, rotated rx 167.56 ry 24.48 rz -95.21 deg; joints [117.936, 25.531, -37.305, 31.965, -59.6, 41.387]
  MoveL 38 to (497.92, -213.5, 158.32) mm, rotated rx 167.56 ry 24.48 rz -95.21 deg; joints [117.936, 25.531, -37.305, 31.965, -59.6, 41.387]
  Establecer velocidad (50.0 mm/s)
  MoveL 39 to (500.24, -213.5, 142.39) mm, rotated rx 167.56 ry 24.48 rz -95.21 deg; joints [118.041, 26.465, -39.392, 32.619, -57.879, 40.001]
  MoveL 40 to (500.27, -213.5, 126.29) mm, rotated rx 167.56 ry 24.48 rz -95.21 deg; joints [118.043, 27.696, -41.364, 33.314, -56.225, 38.721]
  MoveL 41 to (498.03, -213.5, 110.35) mm, rotated rx 167.56 ry 24.48 rz -95.21 deg; joints [117.941, 29.184, -43.164, 34.026, -54.686, 37.585]
  MoveL 42 to (495.96, -213.5, 102.2) mm, rotated rx 167.56 ry 24.48 rz -95.21 deg; joints [117.849, 30.045, -44.016, 34.394, -53.943, 37.064]
  Establecer velocidad (1000.0 mm/s)
  MoveL 43 to (495.96, -213.5, 102.2) mm, rotated rx 167.56 ry 24.48 rz -95.21 deg; joints [117.849, 30.045, -44.016, 34.394, -53.943, 37.064]
  MoveL 44 to (515.57, -213.5, 200.26) mm, rotated rx 167.56 ry 24.48 rz -95.21 deg; joints [118.754, 20.992, -32.866, 30.56, -63.741, 43.353]
  Establecer velocidad (1000.0 mm/s)
  MoveL 45 to (517.53, -213.5, 256.38) mm, rotated rx 167.56 ry 24.48 rz -95.21 deg; joints [118.847, 17.742, -25.712, 29.024, -69.993, 47.14]
  MoveL 46 to (497.92, -213.5, 158.32) mm, rotated rx 167.56 ry 24.48 rz -95.21 deg; joints [117.936, 25.531, -37.305, 31.965, -59.6, 41.387]
  MoveL 47 to (497.92, -213.5, 158.32) mm, rotated rx 167.56 ry 24.48 rz -95.21 deg; joints [117.936, 25.531, -37.305, 31.965, -59.6, 41.387]
  Establecer velocidad (50.0 mm/s)
  MoveL 48 to (491.38, -213.5, 192.68) mm, rotated rx 167.56 ry 24.48 rz -95.21 deg; joints [117.644, 23.921, -32.71, 30.723, -63.4, 44.339]
  Establecer velocidad (1000.0 mm/s)
  MoveL 49 to (491.38, -213.5, 192.68) mm, rotated rx 167.56 ry 24.48 rz -95.21 deg; joints [117.644, 23.921, -32.71, 30.723, -63.4, 44.339]
  MoveL 50 to (510.99, -213.5, 290.74) mm, rotated rx 167.56 ry 24.48 rz -95.21 deg; joints [118.537, 17.022, -21.019, 28.333, -73.974, 49.77]

--- program platder (robot Fanuc LR Mate 200iD/7L) ---
  Suave(1)
  Establecer velocidad (1000.0 mm/s)
  Est. Ref.: RobotiQ 2F-140 Gripper (Mechanism) Base
  Est. herr: Tool 1
  Mostrar Tool 1
  MoveJ 1 to (290.73, 235.99, 302.4) mm, rotated rx 166.28 ry -34.22 rz -82.17 deg; joints [61.508, 54.356, -0.014, -35.867, -97.6, 119.611]
  MoveL 2 to (290.73, 235.99, 302.4) mm, rotated rx 166.28 ry -34.22 rz -82.17 deg; joints [61.508, 54.356, -0.014, -35.867, -97.6, 119.611]
  MoveL 3 to (271.11, 235.99, 204.35) mm, rotated rx 166.28 ry -34.22 rz -82.17 deg; joints [62.142, 58.466, -9.784, -35.608, -89.294, 124.808]
  MoveL 4 to (271.11, 235.99, 204.35) mm, rotated rx 166.28 ry -34.22 rz -82.17 deg; joints [62.142, 58.466, -9.784, -35.608, -89.294, 124.808]
  Establecer velocidad (50.0 mm/s)
  MoveL 5 to (282.7, 237.34, 204.35) mm, rotated rx 166.28 ry -34.22 rz -82.17 deg; joints [61.689, 56.469, -11.551, -35.555, -88.117, 126.199]
  MoveL 6 to (294.36, 237.49, 204.35) mm, rotated rx 166.28 ry -34.22 rz -82.17 deg; joints [61.296, 54.512, -13.249, -35.527, -86.958, 127.499]
  MoveL 7 to (306.01, 237.39, 204.35) mm, rotated rx 166.28 ry -34.22 rz -82.17 deg; joints [60.908, 52.67, -14.817, -35.509, -85.9, 128.719]
  MoveL 8 to (317.63, 236.75, 204.54) mm, rotated rx 166.28 ry -34.22 rz -82.17 deg; joints [60.546, 50.892, -16.275, -35.502, -84.916, 129.853]
  MoveL 9 to (329.71, 235.45, 205.82) mm, rotated rx 166.28 ry -34.22 rz -82.17 deg; joints [60.199, 49.053, -17.601, -35.502, -84.029, 130.898]
  MoveL 10 to (341.48, 233.53, 208.26) mm, rotated rx 166.28 ry -34.22 rz -82.17 deg; joints [59.892, 47.243, -18.708, -35.504, -83.297, 131.783]
  MoveL 11 to (352.97, 231.05, 211.83) mm, rotated rx 166.28 ry -34.22 rz -82.17 deg; joints [59.624, 45.446, -19.608, -35.506, -82.712, 132.518]
  MoveL 12 to (364.33, 228, 215.62) mm, rotated rx 166.28 ry -34.22 rz -82.17 deg; joints [59.39, 43.663, -20.427, -35.512, -82.173, 133.179]
  MoveL 13 to (375.98, 225.17, 218.29) mm, rotated rx 166.28 ry -34.22 rz -82.17 deg; joints [59.122, 41.95, -21.314, -35.519, -81.597, 133.905]
  MoveL 14 to (387.92, 222.97, 219.83) mm, rotated rx 166.28 ry -34.22 rz -82.17 deg; joints [58.792, 40.335, -22.254, -35.519, -81.009, 134.71]
  MoveL 15 to (401.01, 221.36, 220.22) mm, rotated rx 166.28 ry -34.22 rz -82.17 deg; joints [58.365, 38.72, -23.327, -35.508, -80.365, 135.666]
  MoveL 16 to (414.2, 220.57, 220.22) mm, rotated rx 166.28 ry -34.22 rz -82.17 deg; joints [57.863, 37.208, -24.354, -35.475, -79.795, 136.651]
  MoveL 17 to (427.41, 220.48, 220.22) mm, rotated rx 166.28 ry -34.22 rz -82.17 deg; joints [57.296, 35.78, -25.298, -35.415, -79.324, 137.634]
  MoveL 18 to (440.63, 220.48, 220.22) mm, rotated rx 166.28 ry -34.22 rz -82.17 deg; joints [56.704, 34.391, -26.191, -35.341, -78.905, 138.603]
  MoveL 19 to (453.84, 220.48, 220.22) mm, rotated rx 166.28 ry -34.22 rz -82.17 deg; joints [56.093, 33.031, -27.04, -35.254, -78.528, 139.558]
  MoveL 20 to (486.87, 220.48, 220.22) mm, rotated rx 166.28 ry -34.22 rz -82.17 deg; joints [54.476, 29.749, -28.982, -34.974, -77.76, 141.893]
  MoveL 21 to (492.5, 220.04, 220.22) mm, rotated rx 166.28 ry -34.22 rz -82.17 deg; joints [54.218, 29.173, -29.307, -34.929, -77.623, 142.272]
  MoveL 22 to (498.27, 218.3, 220.22) mm, rotated rx 166.28 ry -34.22 rz -82.17 deg; joints [54.043, 28.498, -29.681, -34.918, -77.403, 142.619]
  MoveL 23 to (503.73, 215.19, 220.22) mm, rotated rx 166.28 ry -34.22 rz -82.17 deg; joints [53.981, 27.76, -30.082, -34.949, -77.105, 142.9]
  MoveL 24 to (508.4, 210.82, 220.22) mm, rotated rx 166.28 ry -34.22 rz -82.17 deg; joints [54.053, 27.014, -30.479, -35.027, -76.745, 143.081]
  MoveL 25 to (511.89, 205.55, 220.22) mm, rotated rx 166.28 ry -34.22 rz -82.17 deg; joints [54.257, 26.321, -30.84, -35.146, -76.348, 143.147]
  MoveL 26 to (514.01, 199.84, 220.22) mm, rotated rx 166.28 ry -34.22 rz -82.17 deg; joints [54.572, 25.731, -31.141, -35.296, -75.947, 143.099]
  MoveL 27 to (514.8, 194.16, 220.22) mm, rotated rx 166.28 ry -34.22 rz -82.17 deg; joints [54.96, 25.274, -31.37, -35.463, -75.567, 142.956]
  MoveL 28 to (514.82, 188.65, 220.22) mm, rotated rx 166.28 ry -34.22 rz -82.17 deg; joints [55.382, 24.907, -31.552, -35.634, -75.21, 142.763]
  MoveL 29 to (514.8, 183.15, 220.22) mm, rotated rx 166.28 ry -34.22 rz -82.17 deg; joints [55.81, 24.547, -31.728, -35.807, -74.855, 142.564]
  MoveL 30 to (513.97, 177.46, 220.22) mm, rotated rx 166.28 ry -34.22 rz -82.17 deg; joints [56.298, 24.258, -31.868, -35.995, -74.498, 142.3]
  MoveL 31 to (511.81, 171.76, 220.22) mm, rotated rx 166.28 ry -34.22 rz -82.17 deg; joints [56.862, 24.103, -31.943, -36.197, -74.156, 141.944]
  MoveL 32 to (508.28, 166.5, 220.22) mm, rotated rx 166.28 ry -34.22 rz -82.17 deg; joints [57.461, 24.117, -31.936, -36.395, -73.86, 141.514]
  MoveL 33 to (503.59, 162.17, 220.22) mm, rotated rx 166.28 ry -34.22 rz -82.17 deg; joints [58.045, 24.309, -31.844, -36.571, -73.64, 141.041]
  MoveL 34 to (498.11, 159.09, 220.22) mm, rotated rx 166.28 ry -34.22 rz -82.17 deg; joints [58.563, 24.662, -31.672, -36.71, -73.514, 140.566]
  MoveL 35 to (491.52, 157.26, 220.22) mm, rotated rx 166.28 ry -34.22 rz -82.17 deg; joints [59.029, 25.208, -31.403, -36.812, -73.492, 140.066]
  MoveL 36 to (485.14, 156.98, 220.22) mm, rotated rx 166.28 ry -34.22 rz -82.17 deg; joints [59.355, 25.83, -31.091, -36.859, -73.575, 139.638]
  MoveL 37 to (478.85, 156.98, 220.22) mm, rotated rx 166.28 ry -34.22 rz -82.17 deg; joints [59.649, 26.463, -30.766, -36.894, -73.684, 139.225]
  MoveL 38 to (472.56, 156.98, 220.22) mm, rotated rx 166.28 ry -34.22 rz -82.17 deg; joints [59.938, 27.101, -30.433, -36.925, -73.801, 138.809]
  MoveL 39 to (466.27, 156.98, 220.22) mm, rotated rx 166.28 ry -34.22 rz -82.17 deg; joints [60.222, 27.742, -30.091, -36.952, -73.926, 138.391]
  MoveL 40 to (459.98, 156.98, 220.22) mm, rotated rx 166.28 ry -34.22 rz -82.17 deg; joints [60.501, 28.388, -29.741, -36.975, -74.061, 137.971]
  MoveL 41 to (453.69, 156.98, 220.22) mm, rotated rx 166.28 ry -34.22 rz -82.17 deg; joints [60.776, 29.037, -29.382, -36.995, -74.204, 137.549]
  MoveL 42 to (439.15, 156.98, 220.22) mm, rotated rx 166.28 ry -34.22 rz -82.17 deg; joints [61.392, 30.556, -28.519, -37.028, -74.569, 136.562]
  MoveL 43 to (424.62, 156.98, 220.22) mm, rotated rx 166.28 ry -34.22 rz -82.17 deg; joints [61.985, 32.101, -27.605, -37.043, -74.983, 135.559]
  MoveL 44 to (410.09, 157.19, 220.22) mm, rotated rx 166.28 ry -34.22 rz -82.17 deg; joints [62.54, 33.689, -26.632, -37.037, -75.462, 134.545]
  MoveL 45 to (395.56, 156.87, 220.2) mm, rotated rx 166.28 ry -34.22 rz -82.17 deg; joints [63.113, 35.282, -25.624, -37.03, -75.957, 133.494]
  MoveL 46 to (383.35, 155.91, 219.38) mm, rotated rx 166.28 ry -34.22 rz -82.17 deg; joints [63.628, 36.648, -24.848, -37.043, -76.295, 132.63]
  MoveL 47 to (371.43, 154.37, 217.39) mm, rotated rx 166.28 ry -34.22 rz -82.17 deg; joints [64.161, 38.03, -24.207, -37.077, -76.515, 131.835]
  MoveL 48 to (359.79, 152.27, 214.24) mm, rotated rx 166.28 ry -34.22 rz -82.17 deg; joints [64.709, 39.424, -23.696, -37.13, -76.621, 131.107]
  MoveL 49 to (348.39, 149.63, 210.26) mm, rotated rx 166.28 ry -34.22 rz -82.17 deg; joints [65.273, 40.824, -23.274, -37.197, -76.645, 130.421]
  MoveL 50 to (336.92, 146.37, 207.17) mm, rotated rx 166.28 ry -34.22 rz -82.17 deg; joints [65.868, 42.185, -22.724, -37.247, -76.751, 129.631]
  MoveL 51 to (325.37, 142.49, 205.22) mm, rotated rx 166.28 ry -34.22 rz -82.17 deg; joints [66.495, 43.505, -22.018, -37.278, -76.962, 128.718]
  MoveL 52 to (312.67, 138.92, 204.36) mm, rotated rx 166.28 ry -34.22 rz -82.17 deg; joints [67.118, 44.986, -21.014, -37.264, -77.409, 127.621]
  MoveL 53 to (299.63, 136.58, 204.35) mm, rotated rx 166.28 ry -34.22 rz -82.17 deg; joints [67.651, 46.602, -19.761, -37.199, -78.105, 126.438]
  MoveL 54 to (286.38, 135.5, 204.35) mm, rotated rx 166.28 ry -34.22 rz -82.17 deg; joints [68.089, 48.392, -18.339, -37.101, -78.988, 125.226]
  MoveL 55 to (273.09, 135.71, 204.35) mm, rotated rx 166.28 ry -34.22 rz -82.17 deg; joints [68.43, 50.357, -16.742, -36.978, -80.067, 123.984]
  MoveL 56 to (259.94, 137.19, 204.41) mm, rotated rx 166.28 ry -34.22 rz -82.17 deg; joints [68.673, 52.498, -14.953, -36.838, -81.358, 122.705]
  MoveL 57 to (251.88, 138.75, 204.76) mm, rotated rx 166.28 ry -34.22 rz -82.17 deg; joints [68.777, 53.921, -13.698, -36.744, -82.302, 121.865]
  MoveL 58 to (243.94, 140.77, 205.39) mm, rotated rx 166.28 ry -34.22 rz -82.17 deg; joints [68.845, 55.424, -12.317, -36.649, -83.37, 120.98]
  MoveL 59 to (236.14, 143.27, 206.3) mm, rotated rx 166.28 ry -34.22 rz -82.17 deg; joints [68.878, 57.029, -10.79, -36.557, -84.576, 120.038]
  MoveL 60 to (228.76, 146.69, 207.42) mm, rotated rx 166.28 ry -34.22 rz -82.17 deg; joints [68.842, 58.745, -9.114, -36.47, -85.944, 119.066]
  MoveL 61 to (222.19, 151.5, 208.64) mm, rotated rx 166.28 ry -34.22 rz -82.17 deg; joints [68.7, 60.565, -7.306, -36.395, -87.483, 118.104]
  MoveL 62 to (216.73, 157.49, 209.81) mm, rotated rx 166.28 ry -34.22 rz -82.17 deg; joints [68.46, 62.445, -5.421, -36.341, -89.142, 117.178]
  MoveL 63 to (212.53, 164.51, 210.81) mm, rotated rx 166.28 ry -34.22 rz -82.17 deg; joints [68.131, 64.356, -3.501, -36.315, -90.883, 116.304]
  MoveL 64 to (209.81, 172.2, 211.5) mm, rotated rx 166.28 ry -34.22 rz -82.17 deg; joints [67.729, 66.203, -1.654, -36.321, -92.609, 115.534]
  MoveL 65 to (208.86, 177.63, 211.75) mm, rotated rx 166.28 ry -34.22 rz -82.17 deg; joints [67.424, 67.353, -0.514, -36.339, -93.708, 115.104]
  MoveL 66 to (208.64, 183.15, 211.81) mm, rotated rx 166.28 ry -34.22 rz -82.17 deg; joints [67.098, 68.37, 0.481, -36.363, -94.703, 114.776]
  MoveL 67 to (208.73, 188.67, 211.79) mm, rotated rx 166.28 ry -34.22 rz -82.17 deg; joints [66.765, 69.384, 1.469, -36.397, -95.696, 114.456]
  MoveL 68 to (209.75, 194.03, 211.52) mm, rotated rx 166.28 ry -34.22 rz -82.17 deg; joints [66.418, 70.015, 2.054, -36.415, -96.373, 114.388]
  MoveL 69 to (212.8, 200.65, 210.74) mm, rotated rx 166.28 ry -34.22 rz -82.17 deg; joints [65.945, 69.897, 1.832, -36.374, -96.474, 114.904]
  MoveL 70 to (217.37, 206.3, 209.66) mm, rotated rx 166.28 ry -34.22 rz -82.17 deg; joints [65.488, 68.891, 0.696, -36.271, -95.83, 115.95]
  MoveL 71 to (222.43, 211.45, 208.59) mm, rotated rx 166.28 ry -34.22 rz -82.17 deg; joints [65.045, 67.755, -0.557, -36.167, -95.081, 117.053]
  MoveL 72 to (230.71, 218.41, 207.1) mm, rotated rx 166.28 ry -34.22 rz -82.17 deg; joints [64.401, 65.996, -2.451, -36.021, -93.929, 118.694]
  MoveL 73 to (239.81, 224.45, 205.84) mm, rotated rx 166.28 ry -34.22 rz -82.17 deg; joints [63.782, 64.177, -4.345, -35.89, -92.759, 120.309]
  MoveL 74 to (249.55, 229.41, 204.92) mm, rotated rx 166.28 ry -34.22 rz -82.17 deg; joints [63.199, 62.33, -6.193, -35.778, -91.6, 121.862]
  MoveL 75 to (259.79, 233.23, 204.42) mm, rotated rx 166.28 ry -34.22 rz -82.17 deg; joints [62.661, 60.466, -7.971, -35.685, -90.469, 123.334]
  Establecer velocidad (1000.0 mm/s)
  MoveL 76 to (259.79, 233.23, 204.42) mm, rotated rx 166.28 ry -34.22 rz -82.17 deg; joints [62.661, 60.466, -7.971, -35.685, -90.469, 123.334]
  MoveL 77 to (279.4, 233.23, 302.47) mm, rotated rx 166.28 ry -34.22 rz -82.17 deg; joints [62.044, 56.699, 2.022, -36.094, -98.933, 117.963]
  Establecer velocidad (1000.0 mm/s)
  MoveL 78 to (473.61, 220.65, 367.18) mm, rotated rx 166.28 ry -34.22 rz -82.17 deg; joints [55.128, 26.158, -10.053, -34.28, -93.035, 130.625]
  MoveL 79 to (453.99, 220.65, 269.13) mm, rotated rx 166.28 ry -34.22 rz -82.17 deg; joints [56.074, 30.861, -21.26, -34.717, -83.275, 136.217]
  MoveL 80 to (453.99, 220.65, 269.13) mm, rotated rx 166.28 ry -34.22 rz -82.17 deg; joints [56.074, 30.861, -21.26, -34.717, -83.275, 136.217]
  Establecer velocidad (50.0 mm/s)
  MoveL 81 to (473.84, 219.7, 269.13) mm, rotated rx 166.28 ry -34.22 rz -82.17 deg; joints [55.184, 28.702, -22.431, -34.551, -82.78, 137.572]
  MoveL 82 to (493.53, 216.95, 269.13) mm, rotated rx 166.28 ry -34.22 rz -82.17 deg; joints [54.386, 26.487, -23.559, -34.402, -82.266, 138.827]
  MoveL 83 to (499.94, 215.22, 269.13) mm, rotated rx 166.28 ry -34.22 rz -82.17 deg; joints [54.178, 25.715, -23.934, -34.369, -82.065, 139.199]
  MoveL 84 to (505.78, 212.13, 269.13) mm, rotated rx 166.28 ry -34.22 rz -82.17 deg; joints [54.096, 24.908, -24.316, -34.375, -81.792, 139.48]
  MoveL 85 to (510.85, 207.86, 269.13) mm, rotated rx 166.28 ry -34.22 rz -82.17 deg; joints [54.141, 24.095, -24.69, -34.419, -81.46, 139.659]
  MoveL 86 to (514.84, 202.58, 269.13) mm, rotated rx 166.28 ry -34.22 rz -82.17 deg; joints [54.32, 23.319, -25.036, -34.504, -81.082, 139.722]
  MoveL 87 to (517.37, 196.47, 269.13) mm, rotated rx 166.28 ry -34.22 rz -82.17 deg; joints [54.646, 22.635, -25.334, -34.631, -80.67, 139.647]
  MoveL 88 to (518.11, 189.9, 269.13) mm, rotated rx 166.28 ry -34.22 rz -82.17 deg; joints [55.11, 22.1, -25.561, -34.794, -80.245, 139.429]
  MoveL 89 to (517.79, 183.32, 269.13) mm, rotated rx 166.28 ry -34.22 rz -82.17 deg; joints [55.637, 21.677, -25.737, -34.972, -79.828, 139.135]
  MoveL 90 to (515.9, 177.05, 269.13) mm, rotated rx 166.28 ry -34.22 rz -82.17 deg; joints [56.229, 21.44, -25.834, -35.16, -79.442, 138.748]
  MoveL 91 to (512.43, 171.45, 269.13) mm, rotated rx 166.28 ry -34.22 rz -82.17 deg; joints [56.854, 21.417, -25.844, -35.346, -79.11, 138.287]
  MoveL 92 to (507.82, 166.76, 269.13) mm, rotated rx 166.28 ry -34.22 rz -82.17 deg; joints [57.464, 21.579, -25.777, -35.517, -78.846, 137.792]
  MoveL 93 to (502.49, 163.24, 269.13) mm, rotated rx 166.28 ry -34.22 rz -82.17 deg; joints [58.014, 21.899, -25.645, -35.66, -78.665, 137.301]
  MoveL 94 to (496.51, 160.97, 269.13) mm, rotated rx 166.28 ry -34.22 rz -82.17 deg; joints [58.49, 22.373, -25.445, -35.772, -78.576, 136.827]
  MoveL 95 to (490.27, 159.84, 269.13) mm, rotated rx 166.28 ry -34.22 rz -82.17 deg; joints [58.884, 22.952, -25.197, -35.853, -78.57, 136.385]
  MoveL 96 to (483.98, 158.92, 269.13) mm, rotated rx 166.28 ry -34.22 rz -82.17 deg; joints [59.255, 23.554, -24.932, -35.924, -78.587, 135.948]
  MoveL 97 to (467.87, 157.39, 269.13) mm, rotated rx 166.28 ry -34.22 rz -82.17 deg; joints [60.118, 25.169, -24.193, -36.068, -78.724, 134.858]
  MoveL 98 to (451.69, 156.96, 269.13) mm, rotated rx 166.28 ry -34.22 rz -82.17 deg; joints [60.863, 26.889, -23.36, -36.163, -78.995, 133.796]
  MoveL 99 to (436.98, 157.39, 269.13) mm, rotated rx 166.28 ry -34.22 rz -82.17 deg; joints [61.45, 28.532, -22.52, -36.213, -79.353, 132.847]
  MoveL 100 to (422.43, 159.01, 269.13) mm, rotated rx 166.28 ry -34.22 rz -82.17 deg; joints [61.92, 30.259, -21.593, -36.225, -79.844, 131.933]
  MoveL 101 to (408.16, 161.71, 269.13) mm, rotated rx 166.28 ry -34.22 rz -82.17 deg; joints [62.28, 32.053, -20.584, -36.204, -80.46, 131.052]
  MoveL 102 to (393.62, 161.55, 269.13) mm, rotated rx 166.28 ry -34.22 rz -82.17 deg; joints [62.843, 33.743, -19.59, -36.231, -80.949, 130.025]
  MoveL 103 to (379.08, 161.47, 269.13) mm, rotated rx 166.28 ry -34.22 rz -82.17 deg; joints [63.38, 35.483, -18.525, -36.246, -81.508, 128.973]
  MoveL 104 to (374.76, 161.58, 269.13) mm, rotated rx 166.28 ry -34.22 rz -82.17 deg; joints [63.527, 36.018, -18.19, -36.247, -81.696, 128.659]
  MoveL 105 to (370.45, 161.79, 269.13) mm, rotated rx 166.28 ry -34.22 rz -82.17 deg; joints [63.665, 36.564, -17.843, -36.245, -81.898, 128.346]
  MoveL 106 to (366.14, 162.16, 269.13) mm, rotated rx 166.28 ry -34.22 rz -82.17 deg; joints [63.789, 37.123, -17.484, -36.239, -82.118, 128.035]
  MoveL 107 to (361.88, 162.86, 269.13) mm, rotated rx 166.28 ry -34.22 rz -82.17 deg; joints [63.887, 37.702, -17.108, -36.228, -82.366, 127.734]
  MoveL 108 to (358.11, 164.91, 269.13) mm, rotated rx 166.28 ry -34.22 rz -82.17 deg; joints [63.873, 38.309, -16.709, -36.194, -82.696, 127.508]
  MoveL 109 to (355.65, 167.54, 269.13) mm, rotated rx 166.28 ry -34.22 rz -82.17 deg; joints [63.774, 38.789, -16.39, -36.152, -83.01, 127.395]
  MoveL 110 to (354.04, 170.76, 269.13) mm, rotated rx 166.28 ry -34.22 rz -82.17 deg; joints [63.606, 39.201, -16.113, -36.101, -83.328, 127.362]
  MoveL 111 to (353.58, 174.31, 269.13) mm, rotated rx 166.28 ry -34.22 rz -82.17 deg; joints [63.376, 39.491, -15.918, -36.045, -83.616, 127.426]
  MoveL 112 to (354.33, 177.83, 269.13) mm, rotated rx 166.28 ry -34.22 rz -82.17 deg; joints [63.108, 39.623, -15.828, -35.989, -83.84, 127.583]
  MoveL 113 to (355.49, 181.27, 269.13) mm, rotated rx 166.28 ry -34.22 rz -82.17 deg; joints [62.832, 39.701, -15.775, -35.933, -84.039, 127.768]
  MoveL 114 to (356.66, 184.7, 269.13) mm, rotated rx 166.28 ry -34.22 rz -82.17 deg; joints [62.556, 39.778, -15.723, -35.877, -84.237, 127.953]
  MoveL 115 to (356.99, 187.44, 269.13) mm, rotated rx 166.28 ry -34.22 rz -82.17 deg; joints [62.357, 39.921, -15.626, -35.833, -84.428, 128.052]
  MoveL 116 to (356.16, 190.22, 269.13) mm, rotated rx 166.28 ry -34.22 rz -82.17 deg; joints [62.198, 40.218, -15.423, -35.791, -84.682, 128.057]
  MoveL 117 to (355.36, 193.01, 269.13) mm, rotated rx 166.28 ry -34.22 rz -82.17 deg; joints [62.039, 40.515, -15.218, -35.749, -84.938, 128.063]
  MoveL 118 to (354.57, 195.8, 269.13) mm, rotated rx 166.28 ry -34.22 rz -82.17 deg; joints [61.879, 40.813, -15.012, -35.708, -85.195, 128.067]
  MoveL 119 to (353.84, 198.6, 269.13) mm, rotated rx 166.28 ry -34.22 rz -82.17 deg; joints [61.718, 41.107, -14.808, -35.667, -85.452, 128.075]
  MoveL 120 to (353.78, 203.42, 269.13) mm, rotated rx 166.28 ry -34.22 rz -82.17 deg; joints [61.399, 41.458, -14.562, -35.594, -85.832, 128.183]
  MoveL 121 to (355.4, 207.97, 269.13) mm, rotated rx 166.28 ry -34.22 rz -82.17 deg; joints [61.038, 41.575, -14.481, -35.521, -86.101, 128.42]
  MoveL 122 to (358.25, 211.87, 269.13) mm, rotated rx 166.28 ry -34.22 rz -82.17 deg; joints [60.674, 41.486, -14.543, -35.451, -86.255, 128.744]
  MoveL 123 to (361.5, 214.45, 269.13) mm, rotated rx 166.28 ry -34.22 rz -82.17 deg; joints [60.383, 41.252, -14.707, -35.399, -86.284, 129.069]
  MoveL 124 to (365.46, 215.69, 269.13) mm, rotated rx 166.28 ry -34.22 rz -82.17 deg; joints [60.152, 40.829, -15.002, -35.363, -86.174, 129.423]
  MoveL 125 to (369.63, 216.25, 269.13) mm, rotated rx 166.28 ry -34.22 rz -82.17 deg; joints [59.957, 40.336, -15.342, -35.336, -86.005, 129.774]
  MoveL 126 to (373.81, 216.59, 269.13) mm, rotated rx 166.28 ry -34.22 rz -82.17 deg; joints [59.773, 39.829, -15.689, -35.311, -85.824, 130.12]
  MoveL 127 to (378, 216.76, 269.13) mm, rotated rx 166.28 ry -34.22 rz -82.17 deg; joints [59.599, 39.316, -16.037, -35.289, -85.637, 130.458]
  MoveL 128 to (382.19, 216.81, 269.13) mm, rotated rx 166.28 ry -34.22 rz -82.17 deg; joints [59.431, 38.8, -16.383, -35.268, -85.447, 130.791]
  MoveL 129 to (386.38, 216.77, 269.13) mm, rotated rx 166.28 ry -34.22 rz -82.17 deg; joints [59.268, 38.283, -16.726, -35.248, -85.258, 131.118]
  MoveL 130 to (394.98, 216.55, 269.13) mm, rotated rx 166.28 ry -34.22 rz -82.17 deg; joints [58.937, 37.227, -17.417, -35.207, -84.876, 131.778]
  MoveL 131 to (403.58, 216.27, 269.13) mm, rotated rx 166.28 ry -34.22 rz -82.17 deg; joints [58.602, 36.187, -18.083, -35.165, -84.515, 132.424]
  MoveL 132 to (412.13, 216.76, 269.13) mm, rotated rx 166.28 ry -34.22 rz -82.17 deg; joints [58.211, 35.228, -18.685, -35.106, -84.237, 133.077]
  MoveL 133 to (420.73, 218.78, 269.13) mm, rotated rx 166.28 ry -34.22 rz -82.17 deg; joints [57.705, 34.389, -19.2, -35.012, -84.09, 133.769]
  MoveL 134 to (425.94, 219.88, 269.13) mm, rotated rx 166.28 ry -34.22 rz -82.17 deg; joints [57.402, 33.879, -19.509, -34.954, -84.001, 134.182]
  MoveL 135 to (430.07, 220.4, 269.13) mm, rotated rx 166.28 ry -34.22 rz -82.17 deg; joints [57.184, 33.455, -19.763, -34.914, -83.91, 134.498]
  MoveL 136 to (433.25, 220.6, 269.13) mm, rotated rx 166.28 ry -34.22 rz -82.17 deg; joints [57.028, 33.116, -19.964, -34.887, -83.829, 134.734]
  MoveL 137 to (435.99, 220.65, 269.13) mm, rotated rx 166.28 ry -34.22 rz -82.17 deg; joints [56.902, 32.817, -20.14, -34.865, -83.752, 134.934]
  MoveL 138 to (438.85, 220.65, 269.13) mm, rotated rx 166.28 ry -34.22 rz -82.17 deg; joints [56.773, 32.502, -20.324, -34.843, -83.67, 135.139]
  MoveL 139 to (441.62, 220.65, 269.13) mm, rotated rx 166.28 ry -34.22 rz -82.17 deg; joints [56.647, 32.198, -20.5, -34.821, -83.593, 135.338]
  MoveL 140 to (445.2, 220.65, 269.13) mm, rotated rx 166.28 ry -34.22 rz -82.17 deg; joints [56.483, 31.809, -20.725, -34.792, -83.497, 135.594]
  MoveL 141 to (449.49, 220.65, 269.13) mm, rotated rx 166.28 ry -34.22 rz -82.17 deg; joints [56.284, 31.345, -20.988, -34.756, -83.386, 135.899]
  MoveL 142 to (453.99, 220.65, 269.13) mm, rotated rx 166.28 ry -34.22 rz -82.17 deg; joints [56.074, 30.861, -21.26, -34.717, -83.275, 136.217]
  Establecer velocidad (1000.0 mm/s)
  MoveL 143 to (453.99, 220.65, 269.13) mm, rotated rx 166.28 ry -34.22 rz -82.17 deg; joints [56.074, 30.861, -21.26, -34.717, -83.275, 136.217]
  MoveL 144 to (473.61, 220.65, 367.18) mm, rotated rx 166.28 ry -34.22 rz -82.17 deg; joints [55.128, 26.158, -10.053, -34.28, -93.035, 130.625]

--- program parrder (robot Fanuc LR Mate 200iD/7L) ---
  Suave(1)
  Establecer velocidad (1000.0 mm/s)
  Est. Ref.: RobotiQ 2F-140 Gripper (Mechanism) Base
  Est. herr: Tool 1
  Mostrar Tool 1
  MoveJ 1 to (294.14, 36.7, 296.46) mm, rotated rx 168.69 ry 0 rz -89.99 deg; joints [86.744, 33.884, -9.121, -0.683, -69.59, 93.431]
  MoveL 2 to (294.14, 36.7, 296.46) mm, rotated rx 168.69 ry 0 rz -89.99 deg; joints [86.744, 33.884, -9.121, -0.683, -69.59, 93.431]
  MoveL 3 to (274.53, 36.7, 198.4) mm, rotated rx 168.69 ry 0 rz -89.99 deg; joints [86.831, 39.07, -19.388, -0.724, -59.322, 93.477]
  MoveL 4 to (274.53, 36.7, 198.4) mm, rotated rx 168.69 ry 0 rz -89.99 deg; joints [86.831, 39.07, -19.388, -0.724, -59.322, 93.477]
  Establecer velocidad (50.0 mm/s)
  MoveL 5 to (272.44, 36.7, 198.21) mm, rotated rx 168.69 ry 0 rz -89.99 deg; joints [86.84, 39.367, -19.213, -0.721, -59.497, 93.464]
  MoveL 6 to (270.34, 36.7, 198.02) mm, rotated rx 168.69 ry 0 rz -89.99 deg; joints [86.849, 39.666, -19.034, -0.718, -59.675, 93.452]
  MoveL 7 to (265.01, 36.7, 197.48) mm, rotated rx 168.69 ry 0 rz -89.99 deg; joints [86.872, 40.433, -18.579, -0.709, -60.131, 93.421]
  MoveL 8 to (252.92, 36.7, 196.02) mm, rotated rx 168.69 ry 0 rz -89.99 deg; joints [86.922, 42.216, -17.52, -0.691, -61.189, 93.352]
  MoveL 9 to (225.62, 36.7, 191.52) mm, rotated rx 168.69 ry 0 rz -89.99 deg; joints [87.028, 46.499, -14.955, -0.652, -63.753, 93.202]
  MoveL 10 to (214.97, 36.7, 189.31) mm, rotated rx 168.69 ry 0 rz -89.99 deg; joints [87.068, 48.285, -13.867, -0.637, -64.839, 93.146]
  MoveL 11 to (209.04, 36.7, 187.96) mm, rotated rx 168.69 ry 0 rz -89.99 deg; joints [87.09, 49.317, -13.233, -0.629, -65.473, 93.115]
  MoveL 12 to (205.72, 36.7, 187.17) mm, rotated rx 168.69 ry 0 rz -89.99 deg; joints [87.102, 49.905, -12.869, -0.625, -65.837, 93.098]
  MoveL 13 to (203.61, 36.7, 186.65) mm, rotated rx 168.69 ry 0 rz -89.99 deg; joints [87.109, 50.283, -12.634, -0.622, -66.072, 93.087]
  MoveL 14 to (201.54, 36.7, 186.06) mm, rotated rx 168.69 ry 0 rz -89.99 deg; joints [87.117, 50.662, -12.407, -0.619, -66.299, 93.076]
  MoveL 15 to (199.36, 36.7, 184) mm, rotated rx 168.69 ry 0 rz -89.99 deg; joints [87.124, 51.096, -12.336, -0.617, -66.37, 93.067]
  MoveL 16 to (198.9, 36.7, 182.55) mm, rotated rx 168.69 ry 0 rz -89.99 deg; joints [87.126, 51.212, -12.44, -0.618, -66.266, 93.067]
  MoveL 17 to (198.86, 36.7, 181.03) mm, rotated rx 168.69 ry 0 rz -89.99 deg; joints [87.126, 51.256, -12.612, -0.618, -66.095, 93.069]
  MoveL 18 to (198.86, 36.7, 174.94) mm, rotated rx 168.69 ry 0 rz -89.99 deg; joints [87.126, 51.411, -13.32, -0.622, -65.387, 93.077]
  MoveL 19 to (198.86, 36.7, 162.78) mm, rotated rx 168.69 ry 0 rz -89.99 deg; joints [87.126, 51.756, -14.71, -0.629, -63.996, 93.094]
  Establecer velocidad (1000.0 mm/s)
  MoveL 20 to (198.86, 36.7, 162.78) mm, rotated rx 168.69 ry 0 rz -89.99 deg; joints [87.126, 51.756, -14.71, -0.629, -63.996, 93.094]
  MoveL 21 to (218.47, 36.7, 260.83) mm, rotated rx 168.69 ry 0 rz -89.99 deg; joints [87.055, 46.596, -5.404, -0.605, -73.302, 93.062]
  Establecer velocidad (1000.0 mm/s)
  MoveL 22 to (294.14, 36.7, 296.46) mm, rotated rx 168.69 ry 0 rz -89.99 deg; joints [86.744, 33.884, -9.121, -0.683, -69.59, 93.431]
  MoveL 23 to (274.53, 36.7, 198.4) mm, rotated rx 168.69 ry 0 rz -89.99 deg; joints [86.831, 39.07, -19.388, -0.724, -59.322, 93.477]
  MoveL 24 to (274.53, 36.7, 198.4) mm, rotated rx 168.69 ry 0 rz -89.99 deg; joints [86.831, 39.07, -19.388, -0.724, -59.322, 93.477]
  Establecer velocidad (50.0 mm/s)
  MoveL 25 to (290.09, 36.7, 200.41) mm, rotated rx 168.69 ry 0 rz -89.99 deg; joints [86.763, 36.878, -20.564, -0.749, -58.147, 93.57]
  MoveL 26 to (305.43, 36.7, 203.7) mm, rotated rx 168.69 ry 0 rz -89.99 deg; joints [86.693, 34.719, -21.471, -0.773, -57.241, 93.661]
  MoveL 27 to (320.47, 36.7, 208.25) mm, rotated rx 168.69 ry 0 rz -89.99 deg; joints [86.621, 32.587, -22.114, -0.796, -56.599, 93.752]
  MoveL 28 to (335.07, 36.7, 214.04) mm, rotated rx 168.69 ry 0 rz -89.99 deg; joints [86.548, 30.488, -22.491, -0.816, -56.223, 93.839]
  MoveL 29 to (352.88, 36.7, 223.12) mm, rotated rx 168.69 ry 0 rz -89.99 deg; joints [86.455, 27.871, -22.593, -0.839, -56.122, 93.944]
  MoveL 30 to (369.63, 36.7, 234.02) mm, rotated rx 168.69 ry 0 rz -89.99 deg; joints [86.362, 25.334, -22.282, -0.858, -56.434, 94.042]
  MoveL 31 to (385.16, 36.7, 246.62) mm, rotated rx 168.69 ry 0 rz -89.99 deg; joints [86.272, 22.905, -21.574, -0.872, -57.143, 94.129]
  MoveL 32 to (399.27, 36.7, 260.77) mm, rotated rx 168.69 ry 0 rz -89.99 deg; joints [86.186, 20.617, -20.492, -0.881, -58.226, 94.204]
  Establecer velocidad (1000.0 mm/s)
  MoveL 33 to (399.27, 36.7, 260.77) mm, rotated rx 168.69 ry 0 rz -89.99 deg; joints [86.186, 20.617, -20.492, -0.881, -58.226, 94.204]
  MoveL 34 to (418.88, 36.7, 358.83) mm, rotated rx 168.69 ry 0 rz -89.99 deg; joints [86.059, 15.893, -8.512, -0.823, -70.207, 94.143]
  Establecer velocidad (1000.0 mm/s)
  MoveL 35 to (520.11, 36.7, 358.83) mm, rotated rx 168.69 ry 0 rz -89.99 deg; joints [85.248, 2.727, -10.739, -1.006, -67.994, 95.037]
  MoveL 36 to (500.5, 36.7, 260.77) mm, rotated rx 168.69 ry 0 rz -89.99 deg; joints [85.431, 8.03, -23.893, -1.097, -54.838, 95.112]
  MoveL 37 to (500.5, 36.7, 260.77) mm, rotated rx 168.69 ry 0 rz -89.99 deg; joints [85.431, 8.03, -23.893, -1.097, -54.838, 95.112]
  Establecer velocidad (50.0 mm/s)
  MoveL 38 to (502.78, 36.7, 247.62) mm, rotated rx 168.69 ry 0 rz -89.99 deg; joints [85.411, 8.346, -25.747, -1.128, -52.985, 95.18]
  MoveL 39 to (505.34, 36.7, 234.52) mm, rotated rx 168.69 ry 0 rz -89.99 deg; joints [85.388, 8.683, -27.61, -1.163, -51.123, 95.253]
  MoveL 40 to (508.02, 36.7, 221.45) mm, rotated rx 168.69 ry 0 rz -89.99 deg; joints [85.363, 9.065, -29.486, -1.202, -49.248, 95.332]
  MoveL 41 to (509.41, 36.7, 208.78) mm, rotated rx 168.69 ry 0 rz -89.99 deg; joints [85.351, 9.638, -31.287, -1.239, -47.447, 95.398]
  MoveL 42 to (509.37, 36.7, 196.07) mm, rotated rx 168.69 ry 0 rz -89.99 deg; joints [85.351, 10.442, -33.07, -1.276, -45.665, 95.451]
  MoveL 43 to (507.91, 36.7, 183.53) mm, rotated rx 168.69 ry 0 rz -89.99 deg; joints [85.365, 11.454, -34.793, -1.311, -43.942, 95.49]
  MoveL 44 to (505.04, 36.7, 171.19) mm, rotated rx 168.69 ry 0 rz -89.99 deg; joints [85.391, 12.662, -36.439, -1.345, -42.295, 95.515]
  Establecer velocidad (1000.0 mm/s)
  MoveL 45 to (505.04, 36.7, 171.19) mm, rotated rx 168.69 ry 0 rz -89.99 deg; joints [85.391, 12.662, -36.439, -1.345, -42.295, 95.515]
  MoveL 46 to (524.65, 36.7, 269.25) mm, rotated rx 168.69 ry 0 rz -89.99 deg; joints [85.205, 4.628, -23.09, -1.14, -55.645, 95.346]

--- program Path5 (robot Fanuc LR Mate 200iD/7L) ---
  Suave(1)
  Establecer velocidad (1000.0 mm/s)
  Est. Ref.: bote cera
  Est. herr: Tool 1
  Mostrar Tool 1
  MoveJ 1 to (444.3, -38.05, 200.48) mm, rotated rx 164.21 ry -43.9 rz -78.89 deg; joints [71.112, 29.406, -36.802, -49.317, -70.299, 138.372]
  MoveL 2 to (444.3, -38.05, 200.48) mm, rotated rx 164.21 ry -43.9 rz -78.89 deg; joints [71.112, 29.406, -36.802, -49.317, -70.299, 138.372]
  MoveL 3 to (424.69, -38.05, 102.43) mm, rotated rx 164.21 ry -43.9 rz -78.89 deg; joints [71.679, 39.022, -46.427, -52.751, -63.906, 146.202]
  MoveL 4 to (424.69, -38.05, 102.43) mm, rotated rx 164.21 ry -43.9 rz -78.89 deg; joints [71.679, 39.022, -46.427, -52.751, -63.906, 146.202]
  Establecer velocidad (50.0 mm/s)
  MoveL 5 to (444.85, -37.09, 102.43) mm, rotated rx 164.21 ry -43.9 rz -78.89 deg; joints [71.013, 37.211, -48.009, -53.023, -63.312, 147.915]
  MoveL 6 to (464.85, -34.29, 102.43) mm, rotated rx 164.21 ry -43.9 rz -78.89 deg; joints [70.146, 35.515, -49.467, -53.137, -62.893, 149.608]
  MoveL 7 to (471.35, -32.49, 102.43) mm, rotated rx 164.21 ry -43.9 rz -78.89 deg; joints [69.773, 35.002, -49.904, -53.106, -62.824, 150.163]
  MoveL 8 to (477.25, -29.29, 102.43) mm, rotated rx 164.21 ry -43.9 rz -78.89 deg; joints [69.289, 34.591, -50.252, -52.974, -62.863, 150.686]
  MoveL 9 to (482.36, -24.9, 102.43) mm, rotated rx 164.21 ry -43.9 rz -78.89 deg; joints [68.716, 34.294, -50.503, -52.747, -63.003, 151.158]
  MoveL 10 to (486.36, -19.47, 102.43) mm, rotated rx 164.21 ry -43.9 rz -78.89 deg; joints [68.084, 34.135, -50.637, -52.437, -63.24, 151.551]
  MoveL 11 to (488.81, -13.22, 102.43) mm, rotated rx 164.21 ry -43.9 rz -78.89 deg; joints [67.433, 34.144, -50.63, -52.057, -63.571, 151.828]
  MoveL 12 to (489.45, -6.56, 102.43) mm, rotated rx 164.21 ry -43.9 rz -78.89 deg; joints [66.815, 34.329, -50.474, -51.638, -63.976, 151.961]
  MoveL 13 to (489.26, -1.21, 102.43) mm, rotated rx 164.21 ry -43.9 rz -78.89 deg; joints [66.348, 34.542, -50.294, -51.301, -64.321, 152.011]
  MoveL 14 to (488.04, 3.92, 102.43) mm, rotated rx 164.21 ry -43.9 rz -78.89 deg; joints [65.944, 34.839, -50.043, -50.974, -64.68, 151.974]
  MoveL 15 to (485.78, 8.74, 102.43) mm, rotated rx 164.21 ry -43.9 rz -78.89 deg; joints [65.613, 35.216, -49.723, -50.668, -65.048, 151.849]
  MoveL 16 to (482.65, 12.98, 102.43) mm, rotated rx 164.21 ry -43.9 rz -78.89 deg; joints [65.37, 35.648, -49.354, -50.399, -65.403, 151.646]
  MoveL 17 to (478.81, 16.64, 102.43) mm, rotated rx 164.21 ry -43.9 rz -78.89 deg; joints [65.208, 36.12, -48.95, -50.166, -65.743, 151.379]
  MoveL 18 to (472.91, 20.37, 102.43) mm, rotated rx 164.21 ry -43.9 rz -78.89 deg; joints [65.124, 36.775, -48.387, -49.926, -66.148, 150.945]
  MoveL 19 to (466.27, 22.56, 102.43) mm, rotated rx 164.21 ry -43.9 rz -78.89 deg; joints [65.197, 37.437, -47.813, -49.774, -66.48, 150.432]
  MoveL 20 to (459.37, 23.71, 102.43) mm, rotated rx 164.21 ry -43.9 rz -78.89 deg; joints [65.365, 38.085, -47.249, -49.68, -66.758, 149.883]
  MoveL 21 to (452.43, 24.65, 102.43) mm, rotated rx 164.21 ry -43.9 rz -78.89 deg; joints [65.548, 38.732, -46.683, -49.595, -67.03, 149.326]
  MoveL 22 to (445.47, 25.37, 102.43) mm, rotated rx 164.21 ry -43.9 rz -78.89 deg; joints [65.745, 39.379, -46.113, -49.518, -67.296, 148.76]
  MoveL 23 to (438.5, 25.89, 102.43) mm, rotated rx 164.21 ry -43.9 rz -78.89 deg; joints [65.955, 40.025, -45.542, -49.449, -67.556, 148.187]
  MoveL 24 to (422.01, 26.31, 102.43) mm, rotated rx 164.21 ry -43.9 rz -78.89 deg; joints [66.498, 41.545, -44.187, -49.311, -68.146, 146.805]
  MoveL 25 to (405.53, 25.72, 102.43) mm, rotated rx 164.21 ry -43.9 rz -78.89 deg; joints [67.095, 43.063, -42.819, -49.201, -68.71, 145.387]
  MoveL 26 to (395.81, 24.68, 102.43) mm, rotated rx 164.21 ry -43.9 rz -78.89 deg; joints [67.489, 43.951, -42.014, -49.157, -69.017, 144.53]
  MoveL 27 to (386.23, 23.03, 102.43) mm, rotated rx 164.21 ry -43.9 rz -78.89 deg; joints [67.914, 44.816, -41.224, -49.133, -69.294, 143.668]
  MoveL 28 to (376.69, 21.52, 102.43) mm, rotated rx 164.21 ry -43.9 rz -78.89 deg; joints [68.318, 45.701, -40.412, -49.091, -69.594, 142.8]
  MoveL 29 to (366.99, 21.63, 102.43) mm, rotated rx 164.21 ry -43.9 rz -78.89 deg; joints [68.596, 46.683, -39.507, -48.967, -70.026, 141.922]
  MoveL 30 to (357.3, 21.78, 102.43) mm, rotated rx 164.21 ry -43.9 rz -78.89 deg; joints [68.865, 47.687, -38.577, -48.836, -70.481, 141.032]
  MoveL 31 to (347.6, 21.76, 102.43) mm, rotated rx 164.21 ry -43.9 rz -78.89 deg; joints [69.139, 48.705, -37.628, -48.705, -70.944, 140.125]
  MoveL 32 to (343.19, 21.63, 102.43) mm, rotated rx 164.21 ry -43.9 rz -78.89 deg; joints [69.27, 49.17, -37.193, -48.649, -71.152, 139.707]
  MoveL 33 to (338.79, 21.37, 102.43) mm, rotated rx 164.21 ry -43.9 rz -78.89 deg; joints [69.409, 49.634, -36.758, -48.597, -71.357, 139.285]
  MoveL 34 to (334.41, 20.93, 102.43) mm, rotated rx 164.21 ry -43.9 rz -78.89 deg; joints [69.558, 50.095, -36.326, -48.551, -71.553, 138.859]
  MoveL 35 to (330.13, 19.88, 102.43) mm, rotated rx 164.21 ry -43.9 rz -78.89 deg; joints [69.748, 50.524, -35.923, -48.529, -71.705, 138.434]
  MoveL 36 to (326.54, 17.33, 102.43) mm, rotated rx 164.21 ry -43.9 rz -78.89 deg; joints [70.024, 50.819, -35.644, -48.572, -71.721, 138.057]
  MoveL 37 to (324.33, 14.38, 102.43) mm, rotated rx 164.21 ry -43.9 rz -78.89 deg; joints [70.293, 50.948, -35.523, -48.65, -71.638, 137.81]
  MoveL 38 to (323.12, 10.9, 102.43) mm, rotated rx 164.21 ry -43.9 rz -78.89 deg; joints [70.572, 50.944, -35.526, -48.764, -71.465, 137.654]
  MoveL 39 to (323.2, 7.23, 102.43) mm, rotated rx 164.21 ry -43.9 rz -78.89 deg; joints [70.834, 50.791, -35.671, -48.905, -71.209, 137.621]
  MoveL 40 to (324.86, 1.95, 102.43) mm, rotated rx 164.21 ry -43.9 rz -78.89 deg; joints [71.173, 50.403, -36.036, -49.137, -70.762, 137.722]
  MoveL 41 to (326.66, -3.27, 102.43) mm, rotated rx 164.21 ry -43.9 rz -78.89 deg; joints [71.509, 50.006, -36.409, -49.373, -70.314, 137.835]
  MoveL 42 to (326.11, -5.62, 102.43) mm, rotated rx 164.21 ry -43.9 rz -78.89 deg; joints [71.693, 49.981, -36.433, -49.454, -70.185, 137.751]
  MoveL 43 to (325.42, -7.98, 102.43) mm, rotated rx 164.21 ry -43.9 rz -78.89 deg; joints [71.882, 49.972, -36.441, -49.533, -70.064, 137.653]
  MoveL 44 to (324.74, -10.34, 102.43) mm, rotated rx 164.21 ry -43.9 rz -78.89 deg; joints [72.071, 49.962, -36.45, -49.612, -69.943, 137.556]
  MoveL 45 to (324.07, -12.71, 102.43) mm, rotated rx 164.21 ry -43.9 rz -78.89 deg; joints [72.26, 49.952, -36.46, -49.691, -69.821, 137.459]
  MoveL 46 to (323.42, -15.07, 102.43) mm, rotated rx 164.21 ry -43.9 rz -78.89 deg; joints [72.448, 49.94, -36.471, -49.77, -69.698, 137.363]
  MoveL 47 to (323.04, -17.48, 102.43) mm, rotated rx 164.21 ry -43.9 rz -78.89 deg; joints [72.634, 49.898, -36.511, -49.855, -69.559, 137.293]
  MoveL 48 to (323.61, -22.3, 102.43) mm, rotated rx 164.21 ry -43.9 rz -78.89 deg; joints [72.975, 49.669, -36.725, -50.054, -69.211, 137.28]
  MoveL 49 to (325.72, -26.67, 102.43) mm, rotated rx 164.21 ry -43.9 rz -78.89 deg; joints [73.251, 49.289, -37.082, -50.271, -68.813, 137.422]
  MoveL 50 to (328.93, -30.32, 102.43) mm, rotated rx 164.21 ry -43.9 rz -78.89 deg; joints [73.451, 48.818, -37.522, -50.485, -68.409, 137.677]
  MoveL 51 to (333.15, -32.7, 102.43) mm, rotated rx 164.21 ry -43.9 rz -78.89 deg; joints [73.536, 48.283, -38.021, -50.674, -68.041, 138.047]
  MoveL 52 to (337.94, -33.49, 102.43) mm, rotated rx 164.21 ry -43.9 rz -78.89 deg; joints [73.489, 47.742, -38.525, -50.813, -67.751, 138.493]
  MoveL 53 to (342.79, -33.94, 102.43) mm, rotated rx 164.21 ry -43.9 rz -78.89 deg; joints [73.413, 47.212, -39.017, -50.938, -67.486, 138.946]
  MoveL 54 to (347.65, -34.15, 102.43) mm, rotated rx 164.21 ry -43.9 rz -78.89 deg; joints [73.319, 46.693, -39.497, -51.053, -67.241, 139.4]
  MoveL 55 to (352.52, -34.2, 102.43) mm, rotated rx 164.21 ry -43.9 rz -78.89 deg; joints [73.21, 46.184, -39.967, -51.16, -67.01, 139.854]
  MoveL 56 to (357.39, -34.15, 102.43) mm, rotated rx 164.21 ry -43.9 rz -78.89 deg; joints [73.092, 45.683, -40.428, -51.262, -66.792, 140.306]
  MoveL 57 to (362.84, -34.01, 102.43) mm, rotated rx 164.21 ry -43.9 rz -78.89 deg; joints [72.952, 45.13, -40.936, -51.37, -66.558, 140.81]
  MoveL 58 to (368.29, -33.82, 102.43) mm, rotated rx 164.21 ry -43.9 rz -78.89 deg; joints [72.806, 44.584, -41.436, -51.474, -66.332, 141.311]
  MoveL 59 to (373.74, -33.65, 102.43) mm, rotated rx 164.21 ry -43.9 rz -78.89 deg; joints [72.659, 44.043, -41.929, -51.576, -66.111, 141.808]
  MoveL 60 to (379.19, -33.53, 102.43) mm, rotated rx 164.21 ry -43.9 rz -78.89 deg; joints [72.514, 43.505, -42.418, -51.679, -65.891, 142.3]
  MoveL 61 to (384.54, -34.56, 102.43) mm, rotated rx 164.21 ry -43.9 rz -78.89 deg; joints [72.461, 42.946, -42.924, -51.834, -65.608, 142.763]
  MoveL 62 to (389.95, -35.87, 102.43) mm, rotated rx 164.21 ry -43.9 rz -78.89 deg; joints [72.429, 42.379, -43.437, -52.002, -65.311, 143.222]
  MoveL 63 to (395.88, -37.2, 102.43) mm, rotated rx 164.21 ry -43.9 rz -78.89 deg; joints [72.385, 41.764, -43.989, -52.183, -64.996, 143.724]
  MoveL 64 to (400.6, -37.81, 102.43) mm, rotated rx 164.21 ry -43.9 rz -78.89 deg; joints [72.312, 41.293, -44.411, -52.303, -64.779, 144.128]
  MoveL 65 to (404.29, -38.02, 102.43) mm, rotated rx 164.21 ry -43.9 rz -78.89 deg; joints [72.232, 40.935, -44.732, -52.384, -64.629, 144.447]
  MoveL 66 to (407.74, -38.05, 102.43) mm, rotated rx 164.21 ry -43.9 rz -78.89 deg; joints [72.143, 40.607, -45.024, -52.449, -64.501, 144.746]
  MoveL 67 to (410.73, -38.05, 102.43) mm, rotated rx 164.21 ry -43.9 rz -78.89 deg; joints [72.063, 40.324, -45.276, -52.504, -64.392, 145.005]
  MoveL 68 to (414.58, -38.05, 102.43) mm, rotated rx 164.21 ry -43.9 rz -78.89 deg; joints [71.959, 39.963, -45.596, -52.574, -64.255, 145.337]
  MoveL 69 to (419.4, -38.05, 102.43) mm, rotated rx 164.21 ry -43.9 rz -78.89 deg; joints [71.826, 39.513, -45.995, -52.659, -64.087, 145.751]
  MoveL 70 to (424.69, -38.05, 102.43) mm, rotated rx 164.21 ry -43.9 rz -78.89 deg; joints [71.679, 39.022, -46.427, -52.751, -63.906, 146.202]
  Establecer velocidad (1000.0 mm/s)
  MoveL 71 to (424.69, -38.05, 102.43) mm, rotated rx 164.21 ry -43.9 rz -78.89 deg; joints [71.679, 39.022, -46.427, -52.751, -63.906, 146.202]
  MoveL 72 to (444.3, -38.05, 200.48) mm, rotated rx 164.21 ry -43.9 rz -78.89 deg; joints [71.112, 29.406, -36.802, -49.317, -70.299, 138.372]
  Establecer velocidad (1000.0 mm/s)
  MoveL 73 to (252.98, 46.93, 135.2) mm, rotated rx 164.21 ry -43.9 rz -78.89 deg; joints [69.838, 59.775, -22.309, -46.109, -80.901, 128.089]
  MoveL 74 to (233.37, 46.93, 37.14) mm, rotated rx 164.21 ry -43.9 rz -78.89 deg; joints [70.294, 69.057, -27.206, -46.932, -77.23, 131.417]
  MoveL 75 to (233.37, 46.93, 37.14) mm, rotated rx 164.21 ry -43.9 rz -78.89 deg; joints [70.294, 69.057, -27.206, -46.932, -77.23, 131.417]
  Establecer velocidad (50.0 mm/s)
  MoveL 76 to (226.02, 45.8, 37.29) mm, rotated rx 164.21 ry -43.9 rz -78.89 deg; joints [70.53, 70.223, -25.955, -46.805, -77.932, 130.334]
  MoveL 77 to (218.79, 44.28, 37.67) mm, rotated rx 164.21 ry -43.9 rz -78.89 deg; joints [70.785, 71.403, -24.657, -46.685, -78.653, 129.207]
  MoveL 78 to (211.66, 42.39, 38.29) mm, rotated rx 164.21 ry -43.9 rz -78.89 deg; joints [71.058, 72.604, -23.306, -46.572, -79.4, 128.033]
  MoveL 79 to (204.63, 40.11, 39.12) mm, rotated rx 164.21 ry -43.9 rz -78.89 deg; joints [71.348, 73.837, -21.892, -46.466, -80.179, 126.803]
  MoveL 80 to (197.94, 37.1, 40.12) mm, rotated rx 164.21 ry -43.9 rz -78.89 deg; joints [71.673, 75.038, -20.491, -46.379, -80.925, 125.562]
  MoveL 81 to (191.9, 32.95, 41.21) mm, rotated rx 164.21 ry -43.9 rz -78.89 deg; joints [72.05, 76.099, -19.226, -46.329, -81.541, 124.388]
  MoveL 82 to (186.69, 27.81, 42.29) mm, rotated rx 164.21 ry -43.9 rz -78.89 deg; joints [72.469, 76.959, -18.176, -46.313, -81.98, 123.344]
  MoveL 83 to (182.45, 21.8, 43.26) mm, rotated rx 164.21 ry -43.9 rz -78.89 deg; joints [72.92, 77.552, -17.419, -46.334, -82.192, 122.492]
  MoveL 84 to (179.34, 15.14, 44.03) mm, rotated rx 164.21 ry -43.9 rz -78.89 deg; joints [73.387, 77.817, -17.035, -46.392, -82.134, 121.901]
  MoveL 85 to (177.45, 7.98, 44.53) mm, rotated rx 164.21 ry -43.9 rz -78.89 deg; joints [73.863, 77.721, -17.067, -46.49, -81.782, 121.608]
  MoveL 86 to (176.87, 0.56, 44.68) mm, rotated rx 164.21 ry -43.9 rz -78.89 deg; joints [74.332, 77.268, -17.519, -46.633, -81.146, 121.628]
  MoveL 87 to (177.09, -6.89, 44.62) mm, rotated rx 164.21 ry -43.9 rz -78.89 deg; joints [74.791, 76.641, -18.182, -46.803, -80.373, 121.813]
  MoveL 88 to (178.76, -13.33, 44.18) mm, rotated rx 164.21 ry -43.9 rz -78.89 deg; joints [75.165, 75.777, -19.145, -47.005, -79.456, 122.282]
  MoveL 89 to (181.97, -19.14, 43.38) mm, rotated rx 164.21 ry -43.9 rz -78.89 deg; joints [75.477, 74.674, -20.412, -47.253, -78.38, 123.024]
  MoveL 90 to (186.28, -24.18, 42.38) mm, rotated rx 164.21 ry -43.9 rz -78.89 deg; joints [75.726, 73.473, -21.809, -47.531, -77.262, 123.916]
  MoveL 91 to (190.93, -28.85, 41.4) mm, rotated rx 164.21 ry -43.9 rz -78.89 deg; joints [75.949, 72.314, -23.163, -47.82, -76.198, 124.801]
  MoveL 92 to (195.87, -33.19, 40.48) mm, rotated rx 164.21 ry -43.9 rz -78.89 deg; joints [76.149, 71.192, -24.473, -48.117, -75.186, 125.679]
  MoveL 93 to (204.78, -39.67, 39.1) mm, rotated rx 164.21 ry -43.9 rz -78.89 deg; joints [76.429, 69.379, -26.579, -48.631, -73.598, 127.14]
  MoveL 94 to (214.45, -45.14, 38.02) mm, rotated rx 164.21 ry -43.9 rz -78.89 deg; joints [76.636, 67.622, -28.59, -49.157, -72.137, 128.599]
  MoveL 95 to (224.64, -49.45, 37.35) mm, rotated rx 164.21 ry -43.9 rz -78.89 deg; joints [76.762, 65.935, -30.473, -49.674, -70.829, 130.031]
  MoveL 96 to (235.32, -52.57, 37.14) mm, rotated rx 164.21 ry -43.9 rz -78.89 deg; joints [76.804, 64.297, -32.239, -50.173, -69.664, 131.443]
  MoveL 97 to (246.3, -54.45, 37.14) mm, rotated rx 164.21 ry -43.9 rz -78.89 deg; joints [76.756, 62.736, -33.895, -50.642, -68.64, 132.836]
  MoveL 98 to (257.43, -55.05, 37.14) mm, rotated rx 164.21 ry -43.9 rz -78.89 deg; joints [76.615, 61.275, -35.449, -51.074, -67.749, 134.212]
  MoveL 99 to (268.56, -55.05, 37.14) mm, rotated rx 164.21 ry -43.9 rz -78.89 deg; joints [76.428, 59.897, -36.918, -51.481, -66.948, 135.557]
  MoveL 100 to (279.7, -54.77, 37.14) mm, rotated rx 164.21 ry -43.9 rz -78.89 deg; joints [76.215, 58.584, -38.32, -51.873, -66.21, 136.869]
  MoveL 101 to (290.74, -53.96, 37.61) mm, rotated rx 164.21 ry -43.9 rz -78.89 deg; joints [75.96, 57.307, -39.608, -52.221, -65.575, 138.116]
  MoveL 102 to (302.83, -52.45, 39.26) mm, rotated rx 164.21 ry -43.9 rz -78.89 deg; joints [75.626, 55.883, -40.857, -52.532, -65.014, 139.376]
  MoveL 103 to (314.62, -50.34, 42.07) mm, rotated rx 164.21 ry -43.9 rz -78.89 deg; joints [75.244, 54.454, -41.908, -52.754, -64.605, 140.491]
  MoveL 104 to (326.12, -47.66, 45.97) mm, rotated rx 164.21 ry -43.9 rz -78.89 deg; joints [74.813, 53.012, -42.769, -52.884, -64.338, 141.465]
  MoveL 105 to (337.66, -44.52, 49.46) mm, rotated rx 164.21 ry -43.9 rz -78.89 deg; joints [74.333, 51.639, -43.611, -52.982, -64.109, 142.446]
  MoveL 106 to (349.5, -41.86, 51.82) mm, rotated rx 164.21 ry -43.9 rz -78.89 deg; joints [73.87, 50.344, -44.555, -53.126, -63.808, 143.508]
  MoveL 107 to (361.64, -39.84, 53.02) mm, rotated rx 164.21 ry -43.9 rz -78.89 deg; joints [73.437, 49.126, -45.614, -53.33, -63.419, 144.659]
  MoveL 108 to (376.22, -38.36, 53.18) mm, rotated rx 164.21 ry -43.9 rz -78.89 deg; joints [72.972, 47.784, -46.986, -53.65, -62.861, 146.11]
  MoveL 109 to (390.88, -37.87, 53.18) mm, rotated rx 164.21 ry -43.9 rz -78.89 deg; joints [72.567, 46.459, -48.37, -54.014, -62.264, 147.549]
  MoveL 110 to (405.54, -37.87, 53.18) mm, rotated rx 164.21 ry -43.9 rz -78.89 deg; joints [72.186, 45.156, -49.733, -54.393, -61.669, 148.967]
  MoveL 111 to (420.2, -37.87, 53.18) mm, rotated rx 164.21 ry -43.9 rz -78.89 deg; joints [71.789, 43.886, -51.062, -54.758, -61.105, 150.368]
  MoveL 112 to (427.61, -37.87, 53.18) mm, rotated rx 164.21 ry -43.9 rz -78.89 deg; joints [71.582, 43.257, -51.722, -54.937, -60.831, 151.07]
  MoveL 113 to (435.01, -37.87, 53.18) mm, rotated rx 164.21 ry -43.9 rz -78.89 deg; joints [71.37, 42.635, -52.374, -55.111, -60.564, 151.769]
  MoveL 114 to (442.42, -37.87, 53.18) mm, rotated rx 164.21 ry -43.9 rz -78.89 deg; joints [71.153, 42.02, -53.019, -55.282, -60.304, 152.464]
  MoveL 115 to (449.82, -37.87, 53.18) mm, rotated rx 164.21 ry -43.9 rz -78.89 deg; joints [70.931, 41.412, -53.657, -55.448, -60.05, 153.156]
  MoveL 116 to (457.23, -37.87, 53.18) mm, rotated rx 164.21 ry -43.9 rz -78.89 deg; joints [70.705, 40.811, -54.289, -55.61, -59.802, 153.845]
  MoveL 117 to (464.82, -37.16, 53.18) mm, rotated rx 164.21 ry -43.9 rz -78.89 deg; joints [70.404, 40.222, -54.909, -55.721, -59.597, 154.552]
  MoveL 118 to (470.62, -35.11, 53.18) mm, rotated rx 164.21 ry -43.9 rz -78.89 deg; joints [70.034, 39.819, -55.332, -55.693, -59.533, 155.095]
  MoveL 119 to (475.99, -31.68, 53.18) mm, rotated rx 164.21 ry -43.9 rz -78.89 deg; joints [69.547, 39.495, -55.674, -55.549, -59.568, 155.603]
  MoveL 120 to (480.48, -27.05, 53.18) mm, rotated rx 164.21 ry -43.9 rz -78.89 deg; joints [68.976, 39.281, -55.899, -55.293, -59.704, 156.029]
  MoveL 121 to (483.72, -21.6, 53.18) mm, rotated rx 164.21 ry -43.9 rz -78.89 deg; joints [68.371, 39.195, -55.99, -54.947, -59.93, 156.34]
  MoveL 122 to (485.57, -15.81, 53.18) mm, rotated rx 164.21 ry -43.9 rz -78.89 deg; joints [67.784, 39.232, -55.951, -54.552, -60.221, 156.522]
  MoveL 123 to (486.12, -10.13, 53.18) mm, rotated rx 164.21 ry -43.9 rz -78.89 deg; joints [67.258, 39.371, -55.804, -54.146, -60.546, 156.582]
  MoveL 124 to (486.12, -4.58, 53.18) mm, rotated rx 164.21 ry -43.9 rz -78.89 deg; joints [66.766, 39.553, -55.613, -53.745, -60.883, 156.592]
  MoveL 125 to (486.03, 0.99, 53.18) mm, rotated rx 164.21 ry -43.9 rz -78.89 deg; joints [66.279, 39.746, -55.41, -53.344, -61.225, 156.593]
  MoveL 126 to (484.93, 6.77, 53.18) mm, rotated rx 164.21 ry -43.9 rz -78.89 deg; joints [65.818, 40.028, -55.113, -52.921, -61.613, 156.502]
  MoveL 127 to (482.47, 12.47, 53.18) mm, rotated rx 164.21 ry -43.9 rz -78.89 deg; joints [65.421, 40.417, -54.704, -52.496, -62.043, 156.289]
  MoveL 128 to (478.65, 17.62, 53.18) mm, rotated rx 164.21 ry -43.9 rz -78.89 deg; joints [65.132, 40.897, -54.2, -52.105, -62.484, 155.955]
  MoveL 129 to (473.72, 21.76, 53.18) mm, rotated rx 164.21 ry -43.9 rz -78.89 deg; joints [64.976, 41.431, -53.638, -51.78, -62.903, 155.521]
  MoveL 130 to (468.1, 24.59, 53.18) mm, rotated rx 164.21 ry -43.9 rz -78.89 deg; joints [64.958, 41.977, -53.065, -51.541, -63.267, 155.024]
  MoveL 131 to (462.27, 26.03, 53.18) mm, rotated rx 164.21 ry -43.9 rz -78.89 deg; joints [65.064, 42.493, -52.524, -51.393, -63.554, 154.506]
  MoveL 132 to (453.87, 26.27, 53.18) mm, rotated rx 164.21 ry -43.9 rz -78.89 deg; joints [65.362, 43.177, -51.807, -51.296, -63.859, 153.754]
  MoveL 133 to (445.53, 26.27, 53.18) mm, rotated rx 164.21 ry -43.9 rz -78.89 deg; joints [65.67, 43.855, -51.096, -51.208, -64.154, 153.004]
  MoveL 134 to (437.2, 26.27, 53.18) mm, rotated rx 164.21 ry -43.9 rz -78.89 deg; joints [65.971, 44.543, -50.375, -51.113, -64.458, 152.248]
  MoveL 135 to (428.87, 26.27, 53.18) mm, rotated rx 164.21 ry -43.9 rz -78.89 deg; joints [66.265, 45.242, -49.644, -51.012, -64.77, 151.488]
  MoveL 136 to (415.54, 26.27, 53.18) mm, rotated rx 164.21 ry -43.9 rz -78.89 deg; joints [66.721, 46.382, -48.452, -50.838, -65.289, 150.259]
  MoveL 137 to (402.22, 26.27, 53.18) mm, rotated rx 164.21 ry -43.9 rz -78.89 deg; joints [67.161, 47.551, -47.231, -50.649, -65.834, 149.014]
  MoveL 138 to (388.89, 26.27, 53.18) mm, rotated rx 164.21 ry -43.9 rz -78.89 deg; joints [67.586, 48.752, -45.977, -50.447, -66.405, 147.753]
  MoveL 139 to (375.56, 26.07, 53.18) mm, rotated rx 164.21 ry -43.9 rz -78.89 deg; joints [68.011, 49.979, -44.697, -50.243, -66.992, 146.472]
  MoveL 140 to (362.24, 26.59, 53.05) mm, rotated rx 164.21 ry -43.9 rz -78.89 deg; joints [68.368, 51.281, -43.362, -49.994, -67.651, 145.184]
  MoveL 141 to (350, 27.72, 51.89) mm, rotated rx 164.21 ry -43.9 rz -78.89 deg; joints [68.638, 52.626, -42.159, -49.754, -68.275, 144.054]
  MoveL 142 to (338.05, 29.44, 49.56) mm, rotated rx 164.21 ry -43.9 rz -78.89 deg; joints [68.849, 54.094, -41.019, -49.513, -68.893, 143.01]
  MoveL 143 to (326.38, 31.7, 46.07) mm, rotated rx 164.21 ry -43.9 rz -78.89 deg; joints [69.007, 55.685, -39.93, -49.272, -69.51, 142.043]
  MoveL 144 to (314.9, 34.53, 42.15) mm, rotated rx 164.21 ry -43.9 rz -78.89 deg; joints [69.117, 57.354, -38.812, -49.011, -70.177, 141.083]
  MoveL 145 to (303.3, 37.99, 39.35) mm, rotated rx 164.21 ry -43.9 rz -78.89 deg; joints [69.183, 59.02, -37.497, -48.69, -71.004, 139.997]
  MoveL 146 to (291.59, 41.93, 37.69) mm, rotated rx 164.21 ry -43.9 rz -78.89 deg; joints [69.217, 60.692, -35.984, -48.326, -71.985, 138.783]
  MoveL 147 to (280.25, 44.89, 37.14) mm, rotated rx 164.21 ry -43.9 rz -78.89 deg; joints [69.306, 62.262, -34.4, -47.989, -72.988, 137.494]
  MoveL 148 to (268.66, 46.89, 37.14) mm, rotated rx 164.21 ry -43.9 rz -78.89 deg; joints [69.462, 63.858, -32.706, -47.678, -74.029, 136.093]
  MoveL 149 to (256.9, 47.9, 37.14) mm, rotated rx 164.21 ry -43.9 rz -78.89 deg; joints [69.682, 65.523, -30.941, -47.399, -75.083, 134.612]
  MoveL 150 to (245.09, 47.92, 37.14) mm, rotated rx 164.21 ry -43.9 rz -78.89 deg; joints [69.961, 67.256, -29.107, -47.151, -76.15, 133.052]
  MoveL 151 to (233.37, 46.93, 37.14) mm, rotated rx 164.21 ry -43.9 rz -78.89 deg; joints [70.294, 69.057, -27.206, -46.932, -77.23, 131.417]
  Establecer velocidad (1000.0 mm/s)
  MoveL 152 to (233.37, 46.93, 37.14) mm, rotated rx 164.21 ry -43.9 rz -78.89 deg; joints [70.294, 69.057, -27.206, -46.932, -77.23, 131.417]
  MoveL 153 to (252.98, 46.93, 135.2) mm, rotated rx 164.21 ry -43.9 rz -78.89 deg; joints [69.838, 59.775, -22.309, -46.109, -80.901, 128.089]
